(* CODESYS project Motion.library
   Version: 2025.10.15.1
   Title: Motion
   DefaultNamespace: Motion
   Placeholder: Motion
   Company: Photara

Project tree, tasks and I/O mapping:
  libraries: Base, * (Photara); Communication, * (Photara); Tc2_MC2, * (Beckhoff Automation GmbH); Tc2_MC2_Drive, * (Beckhoff Automation GmbH); Tc2_Standard, * (Beckhoff Automation GmbH); Tc2_System, * (Beckhoff Automation GmbH); Tc2_Utilities, * (Beckhoff Automation GmbH); Tc3_Module, * (Beckhoff Automation GmbH); TcUnit, * (www.tcunit.org)
  BeckhoffAxis/
    DUTs/
      data type E_WebDriveState
      data type ST_BeckhoffAxisConfiguration
      data type ST_BeckhoffAxisStatus
    GVLs/
      global variables GC_BeckhoffAxis
      global variables GPL_BeckhoffAxis
    POUs/
      function CalculateVirtualDistance [ST]
      function block FB_BeckhoffAxis [ST]: Halt, MoveRelative, MoveVelocity, PowerOff, PowerOn, ResetAxis, SetBrake, SetTension, Stop, _InitializeReferences, _SetCommandPermIntlkConfiguration, _BeckhoffMotionFBs, _CyclicFlags, _EvaluateCompletionConditions, _UpdateComponentStatus, Busy, P_AxisConfiguration, P_AxisReference, P_InTension, P_Powered, P_RotaryAxisStatus, CyclicLogic
      function block FB_WebDrive [ST]: _CalculateRadius, _InitializeChildrenDependencies, CyclicLogic
    Testing/
  ITFs/
    Motion/
      interface I_CompleteAxis: MoveAbsolute
      interface I_RotaryAxis: P_AxisReference, P_RotaryAxisStatus, Halt, MoveRelative, MoveVelocity, PowerOff, PowerOn, ResetAxis, SetBrake, SetTension, Stop
      interface I_RotaryEncoder: Read
  RotaryEncoder/
    DUTs/
      data type ST_RotaryEncoderConfiguration
      data type ST_RotaryEncoderStatus
    GVLs/
      global variables GC_RotaryEncoder
      global variables GPL_RotaryEncoder
    POUs/
      function block FB_RotaryEncoder [ST]: Read, _InitializeReferences, _SetCommandPermIntlkConfiguration, _EvaluateCompletionConditions, _UpdateComponentStatus, CyclicLogic
  Zaber/
    DUTs/
      data type E_MoveDirection
      data type E_MoveType
      data type ST_ArcParameters
      data type ST_AxisKinematics
      data type ST_SinParameters
      data type ST_WaitingForBits
      data type ST_ZaberCommandConfiguration
      data type ST_ZaberConfiguration
      data type ST_ZaberHMI
      data type ST_ZaberInitTableFW744
      data type ST_ZaberReply
      data type ST_ZaberStatus
    GVLs/
      global variables GC_Zaber
      global variables GPL_Zaber
    POUs/
      Functions/
        function F_ExtractAxisNumber [ST]
        function F_ExtractDataField [ST]
        function F_ExtractDeviceAddress [ST]
        function F_ExtractMessageChecksum [ST]
        function F_ExtractMotionStatus [ST]
        function F_ZaberExtractExecutionResult [ST]
        function F_ZaberExtractWarnFaultFlag [ST]
        function F_ZaberSplitReplyTokensEx [ST]
      function block FB_ZaberAxisCmdConfiguration [ST]: _BuildTables, _Initialize, _InitializeChildrenDependencies, _InitializeReferences, FB_Init, GetIndexByCmdSendString, GetIndexByPOUName, P_CommandConfigurations, P_PermIntlkConfigurations, P_ZaberConfiguration, P_ZaberInitTableFW744
      function block FB_ZaberSerialAxis [ST]: comm_en_ipv4_static, io_cancel_schedule, io_set_ao, io_set_ao_schedule, io_set_do, io_set_do_schedule, lockstep_driver_disable, lockstep_driver_enable, lockstep_move_abs, lockstep_move_rel, lockstep_move_sin_stop, lockstep_move_stored, lockstep_move_vel, lockstep_park, lockstep_print, lockstep_set_tolerance, lockstep_setup_disable, lockstep_setup_enable, lockstep_stop, lockstep_unpark, move_index, move_rel, move_sin_stop, move_stored, pvt_buffer_erase, pvt_buffer_print, pvt_call, pvt_fifo, pvt_info, pvt_io_cancel_schedule, pvt_io_set_ao, pvt_io_set_ao_schedule, pvt_io_set_do, pvt_io_set_do_schedule, pvt_point, pvt_setup_disable, pvt_setup_live, pvt_setup_store, scope_add, scope_add_io_ai, scope_add_io_ao, scope_add_io_di, scope_add_io_do, scope_start, set_accel, set_autodetect_coil_mode, set_calibration_type, set_comm_address, set_comm_alert, set_comm_command_packets_max, set_comm_en_ipv4_address, set_comm_en_ipv4_dhcp_enabled, set_comm_en_ipv4_gateway, set_comm_en_ipv4_netmask, set_comm_en_mac, set_comm_en_mdns_enable, set_comm_next_owner, set_comm_packet_size_max, set_comm_protocol, set_comm_rs232_baud, set_comm_word_size_max, set_driver_current_approach, set_driver_current_hold, set_driver_current_max, set_driver_current_run, set_driver_enable_mode, set_driver_enabled, set_driver_temperature, set_get_settings_max, set_ictrl_advance_a, set_ictrl_advance_offset, set_ictrl_afcff_inductance, set_ictrl_afcff_ke, set_ictrl_afcff_ki, set_ictrl_afcff_max, set_ictrl_afcff_ss, set_ictrl_afcff_ss_max, set_ictrl_delay, set_ictrl_ff_kd, set_ictrl_ff_kp, set_ictrl_gain_coldmult, set_ictrl_period, set_ictrl_pi_ki, set_ictrl_pi_kp, set_ictrl_type, set_io_ai_1_fc, set_io_ai_2_fc, set_io_ai_3_fc, set_io_ai_4_fc, set_io_di_port, set_io_do_port, set_knob_dir, set_knob_distance, set_knob_enable, set_knob_maxspeed, set_knob_mode, set_knob_speedprofile, set_limit_approach_maxspeed, set_limit_detect_decelonly, set_limit_detect_maxspeed, set_limit_home_action, set_limit_home_bidirectional, set_limit_home_edge, set_limit_home_offset, set_limit_home_posupdate, set_limit_home_preset, set_limit_home_source, set_limit_home_state, set_limit_home_triggered, set_limit_home_tune, set_limit_home_type, set_limit_home_width, set_limit_max, set_limit_min, set_limit_range_mode, set_lockstep_numgroups, set_maxspeed, set_motion_accel_ramptime, set_motion_accelonly, set_motion_busy, set_motion_decelonly, set_motion_index_dist, set_motion_index_num, set_motion_tracking_ai, set_motion_tracking_dir, set_motion_tracking_ki, set_motion_tracking_kp, set_motion_tracking_limit_max, set_motion_tracking_limit_min, set_motion_tracking_scan_dir, set_motion_tracking_scan_maxspeed, set_motion_tracking_scan_offset, set_motion_tracking_scan_period, set_motion_tracking_scan_signal_valid_delay, set_motion_tracking_scan_tolerance, set_motion_tracking_setpoint, set_motion_tracking_settle_period, set_motion_tracking_settle_tolerance, set_motion_tracking_settle_tolerance_met, set_motion_tracking_settled, set_motion_tracking_signal_valid_di, set_motor_current_max, set_motor_inductance, set_motor_ke, set_motor_phase, set_motor_phase_ratio_div1, set_motor_phase_ratio_div2, set_motor_phase_ratio_mult, set_motor_resistance, set_parking_state, set_peripheral_hw_modified, set_peripheral_id, set_peripheral_id_pending, set_peripheral_serial, set_peripheral_serial_pending, set_pos, set_pvt_numseqs, set_resolution, set_scope_channel_size, set_scope_channel_size_max, set_scope_delay, set_scope_numchannels, set_scope_timebase, set_stream_numbufs, set_stream_numstreams, set_system_access, set_system_axiscount, set_system_led_enable, set_system_serial, set_system_temperature, set_system_uptime, set_system_voltage, set_trigger_numactions, set_trigger_numtriggers, set_user_data_0, set_user_data_1, set_user_data_10, set_user_data_11, set_user_data_12, set_user_data_13, set_user_data_14, set_user_data_15, set_user_data_2, set_user_data_3, set_user_data_4, set_user_data_5, set_user_data_6, set_user_data_7, set_user_data_8, set_user_data_9, set_user_vdata_0, set_user_vdata_1, set_user_vdata_2, set_user_vdata_3, set_vel, set_version, set_version_build, storage_append, storage_exists, storage_get, storage_set, stream_arc, stream_buffer_erase, stream_buffer_print, stream_call, stream_circle, stream_fifo, stream_helix, stream_hold_onloff, stream_info, stream_io_cancel_schedule, stream_io_set_ao, stream_io_set_ao_schedule, stream_io_set_do, stream_io_set_do_schedule, stream_line, stream_set, stream_setup_disable, stream_setup_live, stream_setup_store, stream_wait, stream_wait_io, tools_storepos, trigger_action_command, trigger_action_none, trigger_action_setting, trigger_disable, trigger_enable, trigger_when_io, trigger_when_setting, trigger_when_time, activate, axis_restore, comm_en_ipv4_dhcp, driver_disable, driver_enable, get_accel, get_autodetect_coil_mode, get_calibration_type, get_comm_address, get_comm_alert, get_comm_checksum, get_comm_command_packets_max, get_comm_en_ipv4_address, get_comm_en_ipv4_dhcp_enabled, get_comm_en_ipv4_gateway, get_comm_en_ipv4_netmask, get_comm_en_mac, get_comm_en_mdns_enable, get_comm_next_owner, get_comm_packet_size_max, get_comm_protocol, get_comm_rs232_baud, get_comm_word_size_max, get_device_hw_modified, get_device_id, get_driver_current_approach, get_driver_current_hold, get_driver_current_max, get_driver_current_run, get_driver_enable_mode, get_driver_enabled, get_driver_temperature, get_get_settings_max, get_ictrl_advance_a, get_ictrl_advance_offset, get_ictrl_afcff_inductance, get_ictrl_afcff_ke, get_ictrl_afcff_ki, get_ictrl_afcff_max, get_ictrl_afcff_ss, get_ictrl_afcff_ss_max, get_ictrl_delay, get_ictrl_ff_kd, get_ictrl_ff_kp, get_ictrl_gain_coldmult, get_ictrl_period, get_ictrl_pi_ki, get_ictrl_pi_kp, get_ictrl_type, get_io_ai_1_fc, get_io_ai_2_fc, get_io_ai_3_fc, get_io_ai_4_fc, get_io_di_port, get_io_do_port, get_knob_dir, get_knob_distance, get_knob_enable, get_knob_maxspeed, get_knob_mode, get_knob_speedprofile, get_limit_approach_maxspeed, get_limit_detect_decelonly, get_limit_detect_maxspeed, get_limit_home_action, get_limit_home_bidirectional, get_limit_home_edge, get_limit_home_offset, get_limit_home_posupdate, get_limit_home_preset, get_limit_home_source, get_limit_home_state, get_limit_home_triggered, get_limit_home_tune, get_limit_home_type, get_limit_home_width, get_limit_max, get_limit_min, get_limit_range_mode, get_lockstep_numgroups, get_maxspeed, get_motion_accel_ramptime, get_motion_accelonly, get_motion_busy, get_motion_decelonly, get_motion_index_dist, get_motion_index_num, get_motion_tracking_ai, get_motion_tracking_dir, get_motion_tracking_ki, get_motion_tracking_kp, get_motion_tracking_limit_max, get_motion_tracking_limit_min, get_motion_tracking_scan_dir, get_motion_tracking_scan_maxspeed, get_motion_tracking_scan_offset, get_motion_tracking_scan_period, get_motion_tracking_scan_signal_valid_delay, get_motion_tracking_scan_tolerance, get_motion_tracking_setpoint, get_motion_tracking_settle_period, get_motion_tracking_settle_tolerance, get_motion_tracking_settle_tolerance_met, get_motion_tracking_settled, get_motion_tracking_signal_valid_di, get_motor_current_max, get_motor_inductance, get_motor_ke, get_motor_phase, get_motor_phase_ratio_div1, get_motor_phase_ratio_div2, get_motor_phase_ratio_mult, get_motor_resistance, get_parking_state, get_peripheral_hw_modified, get_peripheral_id, get_peripheral_id_pending, get_peripheral_serial, get_peripheral_serial_pending, get_pos, get_pvt_numseqs, get_resolution, get_scope_channel_size, get_scope_channel_size_max, get_scope_delay, get_scope_numchannels, get_scope_timebase, get_stream_numbufs, get_stream_numstreams, get_system_access, get_system_axiscount, get_system_current_max, get_system_led_enable, get_system_serial, get_system_temperature, get_system_uptime, get_system_voltage, get_trigger_numactions, get_trigger_numtriggers, get_user_data_0, get_user_data_1, get_user_data_10, get_user_data_11, get_user_data_12, get_user_data_13, get_user_data_14, get_user_data_15, get_user_data_2, get_user_data_3, get_user_data_4, get_user_data_5, get_user_data_6, get_user_data_7, get_user_data_8, get_user_data_9, get_user_vdata_0, get_user_vdata_1, get_user_vdata_2, get_user_vdata_3, get_vel, get_version, get_version_build, home, io_get_ai, io_get_ao, io_get_di, io_get_do, io_info, lockstep_get, lockstep_home, lockstep_move_max, lockstep_move_min, lockstep_move_sin, move_abs, move_index_next, move_index_prev, move_max, move_min, move_scan_track_once, move_sin, move_track, move_vel, pvt_buffer_list, renumber, scope_clear, scope_print, scope_stop, set_comm_checksum, stop, storage_erase, storage_print, stream_buffer_list, system_errors, system_factoryreset, system_reset, system_restore, tools_echo, tools_findrange, tools_gotolimit, tools_parking, tools_setcomm, tools_storepos_current, tools_storepos_position, trigger_print, trigger_show, trigger_when_dist, trigger_when_encoder_dist, warnings, warnings_clear, CyclicLogic, P_ZaberConfiguration, _Initialize, _InitializeChildrenDependencies, _InitializeReferences, FB_Init, InjectDependencies, _BuildCommandStringNoArgs, _ClearTempString, _ConfigurationCyclic, _DebugTesting, _DispatchValid, _GetConfigParametersOnInit, _MapIndicesToCommands, _MonitorAsynchronousRequests, _PollBusy, _PopulateStatusStructureWithResponseData, _ReceiveCyclic, _ResolveZaberConfiguration, _ResolveZaberDispatchIndex, _SendCyclic, _TryRehashDispatchIndex, _ExecuteCommandByIndexCyclic, ExecuteCommand, InjectConfigurations, P_I_RingBufferKeyString
      function block FB_ZaberSerialGroup [ST]: _ControllerAxisConfiguration, _Initialize, _InitializeChildrenDependencies, CyclicLogic, FB_Init
    Testing/
      function block FB_ValidateStringHandlingTests [ST]: GivenBusyReplyExpectCorrectFieldExtractionChecksum, GivenBusyReplyExpectCorrectFieldExtractionNoChecksum, GivenIdleReplyExpectCorrectFieldExtractionChecksum, GivenIdleReplyExpectCorrectFieldExtractionChecksum_1, GivenIdleReplyExpectCorrectFieldExtractionNoChecksum, GivenNIReplyExpectCorrectFieldExtractionChecksum, GivenNIReplyExpectCorrectFieldExtractionNoChecksum, GivenReply_ExpectCorrectTokenization
      function block FB_ZaberAxisTests [ST]
      program PRG_TEST [ST]
  program MAIN [ST]
*)

// BeckhoffAxis/DUTs/E_WebDriveState
{attribute 'qualified_only'}
{attribute 'strict'}
{attribute 'to_string'}
TYPE E_WebDriveState :
(
	INIT := 0,
	STOP,
	RESET,
	ERROR,
	IDLE,
	BUSY_TENSION,
	BUSY_SCROLL,
	CALIBRATION
);
END_TYPE

// BeckhoffAxis/DUTs/ST_BeckhoffAxisConfiguration
TYPE ST_BeckhoffAxisConfiguration :
STRUCT
	ComponentConfiguration : REFERENCE TO Base.ST_ComponentConfiguration;
	
	lrTorqueRamp : LREAL := 3; // Tensies per second
	lrMaxSpeed	 : LREAL := 2_000.0; // mm/s
	
	lrScrollVelocity : LREAL := 400.0; // mm/s
END_STRUCT
END_TYPE

// BeckhoffAxis/DUTs/ST_BeckhoffAxisStatus
TYPE ST_BeckhoffAxisStatus :
STRUCT
	BaseComponentStatus : REFERENCE TO Base.ST_ComponentStatus;
	
END_STRUCT
END_TYPE

// RotaryEncoder/DUTs/ST_RotaryEncoderConfiguration
TYPE ST_RotaryEncoderConfiguration :
STRUCT
	ComponentConfiguration : REFERENCE TO Base.ST_ComponentConfiguration;
	CPmm : REAL := 13.123; // clicks on encoder per mm travelled
END_STRUCT
END_TYPE

// RotaryEncoder/DUTs/ST_RotaryEncoderStatus
TYPE ST_RotaryEncoderStatus :
STRUCT
	BaseComponentStatus : REFERENCE TO Base.ST_ComponentStatus;
END_STRUCT
END_TYPE

// Zaber/DUTs/E_MoveDirection
{attribute 'qualified_only'}
{attribute 'strict'}
{attribute 'to_string'}
TYPE E_MoveDirection :
(
	cw := 0, //clockwise
	ccw := 1 //counter-clockwise
);
END_TYPE

// Zaber/DUTs/E_MoveType
{attribute 'qualified_only'}
{attribute 'strict'}
{attribute 'to_string'}
TYPE E_MoveType :
(
	move_abs := 0,
	move_rel := 1
);
END_TYPE

// Zaber/DUTs/ST_ArcParameters
TYPE ST_ArcParameters :
STRUCT
	Axis1 : UINT; //<axis1> The first stream axis on which TO execute the arc segment (optional).  The first stream axis is labelled "a", the second "b", AND so on
	Axis2 : UINT; //<axis2> The second stream axis on which to execute the arc segment (optional). The first stream axis is labelled "a", the second "b", and so on
	MoveType : E_MoveType; //abs Indicates that position parameters are absolute positions; rel Indicates that position parameters are relative to the end point of the previous path segment
	Direction : E_MoveDirection; //cw Indicates that the arc should be in the clockwise direction; //ccw Indicates that the arc should be in the counter-clockwise direction
	CenterX : DINT; //<centrex> The x-axis position of the arc’s centre; Must be the range -2,147,483,648 to 2,147,483,647
	CenterY : DINT; //<centrey> The y-axis position of the arc’s centre; Must be the range -2,147,483,648 to 2,147,483,647
	EndX : DINT; //<endx> The x-axis position of the end of the arc; Must be in the range limit.min to limit.max for that axis
	EndY : DINT; //<endy> The y-axis position of the end of the arc; Must be in the range limit.min to limit.max for that axis
END_STRUCT
END_TYPE

// Zaber/DUTs/ST_AxisKinematics
TYPE ST_AxisKinematics :
STRUCT
	Position	: UDINT;
	Velocity	: DINT;
	Accel		: UDINT;
END_STRUCT
END_TYPE

// Zaber/DUTs/ST_SinParameters
TYPE ST_SinParameters :
STRUCT
	Amplitude					: LREAL := 50000;
	Period						: LREAL := 2000; // ms
	Count						: LREAL := 30;
END_STRUCT
END_TYPE

// Zaber/DUTs/ST_WaitingForBits
TYPE ST_WaitingForBits :
STRUCT
	WaitingForResolution	: BOOL;
	WaitingForMaxSpeed		: BOOL;
END_STRUCT
END_TYPE

// Zaber/DUTs/ST_ZaberCommandConfiguration
TYPE ST_ZaberCommandConfiguration :
STRUCT
 //   CmdIndex			: DINT; 
    PouName 			: STRING;
    CmdDesc				: STRING;
	CmdExecutionType	: Base.E_CommandExecutionType;
END_STRUCT
END_TYPE

// Zaber/DUTs/ST_ZaberConfiguration
TYPE ST_ZaberConfiguration :
STRUCT
	ComponentConfiguration 			: REFERENCE TO ST_ComponentConfiguration;
	ConfiguredComPort				: UDINT := 3;
	ConfiguredTerminationTx			: STRING(5) := '$N';
	ConfiguredTerminationRx			: STRING(5) := '$R$N';
	sControllerRef					: STRING(5) := '/0';
	AxisRef							: UINT := 0;
	MinDynamics						: ST_AxisKinematics;
	MaxDynamics						: ST_AxisKinematics := (Position := 227000, Velocity := 100000, Accel := 15000);
	SetDynamics						: ST_AxisKinematics := (Position := 113000, Velocity := MaxDynamics.Velocity, Accel := MaxDynamics.Accel);
	MaxPollingTime					: TIME := T#50MS;
	MinPollingTime					: TIME := T#5MS;
	EnableSerialInterface			: BOOL := TRUE;
	PollingIntervalTime				: TIME := T#20MS;
	EnablePollingOnMotion			: BOOL := TRUE;
	Resolution						: REAL; // microstep div
	Resolution_um					: REAL := 1.984375; // µm; given by manual
	StreamNumber					: ARRAY[GPL_Zaber.INDEX_STREAM_MIN..GPL_Zaber.INDEX_STREAM_MAX] OF UDINT; 
	BufferNumber					: UDINT;
	LockstepGroup					: USINT := 1;
	TimeConversionFactor			: REAL := 16.384; //s; given by manual
	EnableDynamicPollingInterval	: BOOL := TRUE;
	DefaultPollingTime				: TIME := T#10MS;
	EnableGetParametersOnInit		: BOOL;
	RelativeDistanceMove			: UDINT := 1000; // µm; 
	SinParameters					: ST_SinParameters;
	ArcParameters					: ST_ArcParameters;
	Direction						: BOOL := TRUE; //Right/CW = TRUE
	GetSetting						: STRING(15) := 'twist';
	OptionalValue					: STRING(GPL_Zaber.STRING_LENGTH);
END_STRUCT
END_TYPE

// Zaber/DUTs/ST_ZaberHMI
TYPE ST_ZaberHMI :
STRUCT
    ReplyFlag		: STRING(GPL_Zaber.STRING_LENGTH);  // 'OK' / 'RJ'
    MotionStatus	: BOOL;  // BUSY / IDLE
    WarnFlag    	: STRING(GPL_Zaber.STRING_LENGTH);  // '--' or 'FV'… or 'NI'
    DataField   	: STRING(GPL_Zaber.STRING_LENGTH);  // '0', '12345', etc.
    Checksum    	: STRING(GPL_Zaber.STRING_LENGTH);  // ':CC' or ''
	Footer			: STRING(GPL_Zaber.STRING_LENGTH);
	Position		: DINT;
	Velocity		: DINT; // parsed from Data Field
END_STRUCT
END_TYPE

// Zaber/DUTs/ST_ZaberInitTableFW744
TYPE ST_ZaberInitTableFW744 :
STRUCT
    CmdIndex        : ARRAY[GC_Zaber.INDEX_COMMAND_MIN..GC_Zaber.INDEX_COMMAND_MAX] OF DINT; 
    PouName : ARRAY[GC_Zaber.INDEX_COMMAND_MIN..GC_Zaber.INDEX_COMMAND_MAX] OF STRING := [
        'activate',
        'axis_restore',
        'driver_disable',
        'driver_enable',
        'home',
        'renumber',
        'stop',
        'warnings',
        'comm_en_ipv4_dhcp',
        'comm_en_ipv4_static',
        'io_cancel_schedule',
        'io_get_ai',
        'io_get_ao',
        'io_get_di',
        'io_get_do',
        'io_info',
        'io_set_ao',
        'io_set_ao_schedule',
        'io_set_do',
        'io_set_do_schedule',
        'move_abs',
        'move_index',
        'move_index_next',
        'move_index_prev',
        'move_min',
        'move_max',
        'move_rel',
        'move_scan_track_once',
        'move_sin',
        'move_sin_stop',
        'move_stored',
        'move_track',
        'move_vel',
        'lockstep_driver_disable',
        'lockstep_driver_enable',
        'lockstep_get',
        'lockstep_home',
        'lockstep_move_abs',
        'lockstep_move_min',
        'lockstep_move_max',
        'lockstep_move_rel',
        'lockstep_move_sin',
        'lockstep_move_sin_stop',
        'lockstep_move_stored',
        'lockstep_move_vel',
        'lockstep_park',
        'lockstep_unpark',
        'lockstep_print',
        'lockstep_set_tolerance',
        'lockstep_setup_disable',
        'lockstep_setup_enable',
        'lockstep_stop',
        'pvt_buffer_erase',
        'pvt_buffer_list',
        'pvt_buffer_print',
        'pvt_call',
        'pvt_fifo',
        'pvt_info',
        'pvt_io_cancel_schedule',
        'pvt_io_set_ao',
        'pvt_io_set_ao_schedule',
        'pvt_io_set_do',
        'pvt_io_set_do_schedule',
        'pvt_point',
        'pvt_setup_disable',
        'pvt_setup_live',
        'pvt_setup_store',
        'scope_add',
        'scope_add_io_ai',
        'scope_add_io_ao',
        'scope_add_io_di',
        'scope_add_io_do',
        'scope_clear',
        'scope_print',
        'scope_start',
        'scope_stop',
        'storage_append',
        'storage_erase',
        'storage_exists',
        'storage_get',
        'storage_print',
        'storage_set',
        'stream_arc',
        'stream_buffer_erase',
        'stream_buffer_list',
        'stream_buffer_print',
        'stream_call',
        'stream_circle',
        'stream_fifo',
        'stream_helix',
        'stream_hold_onloff',
        'stream_info',
        'stream_io_cancel_schedule',
        'stream_io_set_ao',
        'stream_io_set_ao_schedule',
        'stream_io_set_do',
        'stream_io_set_do_schedule',
        'stream_line',
        'stream_set',
        'stream_setup_disable',
        'stream_setup_live',
        'stream_setup_store',
        'stream_wait',
        'stream_wait_io',
        'system_errors',
        'system_factoryreset',
        'system_reset',
        'system_restore',
        'tools_echo',
        'tools_findrange',
        'tools_gotolimit',
        'tools_parking',
        'tools_setcomm',
        'tools_storepos',
        'tools_storepos_current',
        'tools_storepos_position',
        'trigger_action_command',
        'trigger_action_none',
        'trigger_action_setting',
        'trigger_disable',
        'trigger_enable',
        'trigger_print',
        'trigger_show',
        'trigger_when_encoder_dist',
        'trigger_when_dist',
        'trigger_when_io',
        'trigger_when_setting',
        'trigger_when_time',
        'get_accel',
        'get_autodetect_coil_mode',
        'get_calibration_type',
        'get_comm_address',
        'get_comm_alert',
        'get_comm_checksum',
        'get_comm_command_packets_max',
        'get_comm_en_ipv4_address',
        'get_comm_en_ipv4_dhcp_enabled',
        'get_comm_en_ipv4_gateway',
        'get_comm_en_ipv4_netmask',
        'get_comm_en_mac',
        'get_comm_en_mdns_enable',
        'get_comm_next_owner',
        'get_comm_packet_size_max',
        'get_comm_protocol',
        'get_comm_rs232_baud',
        'get_comm_word_size_max',
        'get_device_hw_modified',
        'get_device_id',
        'get_driver_current_approach',
        'get_driver_current_hold',
        'get_driver_current_max',
        'get_driver_current_run',
        'get_driver_enable_mode',
        'get_driver_enabled',
        'get_driver_temperature',
        'get_get_settings_max',
        'get_ictrl_advance_a',
        'get_ictrl_advance_offset',
        'get_ictrl_afcff_inductance',
        'get_ictrl_afcff_ke',
        'get_ictrl_afcff_ki',
        'get_ictrl_afcff_max',
        'get_ictrl_afcff_ss',
        'get_ictrl_afcff_ss_max',
        'get_ictrl_delay',
        'get_ictrl_ff_kd',
        'get_ictrl_ff_kp',
        'get_ictrl_gain_coldmult',
        'get_ictrl_period',
        'get_ictrl_pi_ki',
        'get_ictrl_pi_kp',
        'get_ictrl_type',
        'get_io_ai_1_fc',
        'get_io_ai_2_fc',
        'get_io_ai_3_fc',
        'get_io_ai_4_fc',
        'get_io_di_port',
        'get_io_do_port',
        'get_knob_dir',
        'get_knob_distance',
        'get_knob_enable',
        'get_knob_maxspeed',
        'get_knob_mode',
        'get_knob_speedprofile',
        'get_limit_approach_maxspeed',
        'get_limit_detect_decelonly',
        'get_limit_detect_maxspeed',
        'get_limit_home_action',
        'get_limit_home_bidirectional',
        'get_limit_home_edge',
        'get_limit_home_offset',
        'get_limit_home_posupdate',
        'get_limit_home_preset',
        'get_limit_home_source',
        'get_limit_home_state',
        'get_limit_home_triggered',
        'get_limit_home_tune',
        'get_limit_home_type',
        'get_limit_home_width',
        'get_limit_max',
        'get_limit_min',
        'get_limit_range_mode',
        'get_lockstep_numgroups',
        'get_maxspeed',
        'get_motion_accel_ramptime',
        'get_motion_accelonly',
        'get_motion_busy',
        'get_motion_decelonly',
        'get_motion_index_dist',
        'get_motion_index_num',
        'get_motion_tracking_ai',
        'get_motion_tracking_dir',
        'get_motion_tracking_ki',
        'get_motion_tracking_kp',
        'get_motion_tracking_limit_max',
        'get_motion_tracking_limit_min',
        'get_motion_tracking_scan_dir',
        'get_motion_tracking_scan_maxspeed',
        'get_motion_tracking_scan_offset',
        'get_motion_tracking_scan_period',
        'get_motion_tracking_scan_signal_valid_delay',
        'get_motion_tracking_scan_tolerance',
        'get_motion_tracking_setpoint',
        'get_motion_tracking_settle_period',
        'get_motion_tracking_settle_tolerance',
        'get_motion_tracking_settle_tolerance_met',
        'get_motion_tracking_settled',
        'get_motion_tracking_signal_valid_di',
        'get_motor_current_max',
        'get_motor_inductance',
        'get_motor_ke',
        'get_motor_phase',
        'get_motor_phase_ratio_div1',
        'get_motor_phase_ratio_div2',
        'get_motor_phase_ratio_mult',
        'get_motor_resistance',
        'get_parking_state',
        'get_peripheral_hw_modified',
        'get_peripheral_id',
        'get_peripheral_id_pending',
        'get_peripheral_serial',
        'get_peripheral_serial_pending',
        'get_pos',
        'get_pvt_numseqs',
        'get_resolution',
        'get_scope_channel_size',
        'get_scope_channel_size_max',
        'get_scope_delay',
        'get_scope_numchannels',
        'get_scope_timebase',
        'get_stream_numbufs',
        'get_stream_numstreams',
        'get_system_access',
        'get_system_axiscount',
        'get_system_current_max',
        'get_system_led_enable',
        'get_system_serial',
        'get_system_temperature',
        'get_system_uptime',
        'get_system_voltage',
        'get_trigger_numactions',
        'get_trigger_numtriggers',
        'get_user_data_0',
        'get_user_data_1',
        'get_user_data_10',
        'get_user_data_11',
        'get_user_data_12',
        'get_user_data_13',
        'get_user_data_14',
        'get_user_data_15',
        'get_user_data_2',
        'get_user_data_3',
        'get_user_data_4',
        'get_user_data_5',
        'get_user_data_6',
        'get_user_data_7',
        'get_user_data_8',
        'get_user_data_9',
        'get_user_vdata_0',
        'get_user_vdata_1',
        'get_user_vdata_2',
        'get_user_vdata_3',
        'get_vel',
        'get_version',
        'get_version_build',
        'set_accel',
        'set_autodetect_coil_mode',
        'set_calibration_type',
        'set_comm_address',
        'set_comm_alert',
        'set_comm_checksum',
        'set_comm_command_packets_max',
        'set_comm_en_ipv4_address',
        'set_comm_en_ipv4_dhcp_enabled',
        'set_comm_en_ipv4_gateway',
        'set_comm_en_ipv4_netmask',
        'set_comm_en_mdns_enable',
        'set_comm_en_mac',
        'set_comm_next_owner',
        'set_comm_packet_size_max',
        'set_comm_protocol',
        'set_comm_rs232_baud',
        'set_comm_word_size_max',
        'set_driver_current_approach',
        'set_driver_current_hold',
        'set_driver_current_max',
        'set_driver_current_run',
        'set_driver_enable_mode',
        'set_driver_enabled',
        'set_driver_temperature',
        'set_get_settings_max',
        'set_ictrl_advance_a',
        'set_ictrl_advance_offset',
        'set_ictrl_afcff_inductance',
        'set_ictrl_afcff_ke',
        'set_ictrl_afcff_ki',
        'set_ictrl_afcff_max',
        'set_ictrl_afcff_ss',
        'set_ictrl_afcff_ss_max',
        'set_ictrl_delay',
        'set_ictrl_ff_kd',
        'set_ictrl_ff_kp',
        'set_ictrl_gain_coldmult',
        'set_ictrl_period',
        'set_ictrl_pi_ki',
        'set_ictrl_pi_kp',
        'set_ictrl_type',
        'set_io_ai_1_fc',
        'set_io_ai_2_fc',
        'set_io_ai_3_fc',
        'set_io_ai_4_fc',
        'set_io_di_port',
        'set_io_do_port',
        'set_knob_dir',
        'set_knob_distance',
        'set_knob_enable',
        'set_knob_maxspeed',
        'set_knob_mode',
        'set_knob_speedprofile',
        'set_limit_approach_maxspeed',
        'set_limit_detect_decelonly',
        'set_limit_detect_maxspeed',
        'set_limit_home_action',
        'set_limit_home_bidirectional',
        'set_limit_home_edge',
        'set_limit_home_offset',
        'set_limit_home_posupdate',
        'set_limit_home_preset',
        'set_limit_home_source',
        'set_limit_home_state',
        'set_limit_home_triggered',
        'set_limit_home_tune',
        'set_limit_home_type',
        'set_limit_home_width',
        'set_limit_max',
        'set_limit_min',
        'set_limit_range_mode',
        'set_lockstep_numgroups',
        'set_maxspeed',
        'set_motion_accel_ramptime',
        'set_motion_accelonly',
        'set_motion_busy',
        'set_motion_decelonly',
        'set_motion_index_dist',
        'set_motion_index_num',
        'set_motion_tracking_ai',
        'set_motion_tracking_dir',
        'set_motion_tracking_ki',
        'set_motion_tracking_kp',
        'set_motion_tracking_limit_max',
        'set_motion_tracking_limit_min',
        'set_motion_tracking_scan_dir',
        'set_motion_tracking_scan_maxspeed',
        'set_motion_tracking_scan_offset',
        'set_motion_tracking_scan_period',
        'set_motion_tracking_scan_signal_valid_delay',
        'set_motion_tracking_scan_tolerance',
        'set_motion_tracking_setpoint',
        'set_motion_tracking_settle_period',
        'set_motion_tracking_settle_tolerance',
        'set_motion_tracking_settle_tolerance_met',
        'set_motion_tracking_settled',
        'set_motion_tracking_signal_valid_di',
        'set_motor_current_max',
        'set_motor_inductance',
        'set_motor_ke',
        'set_motor_phase',
        'set_motor_phase_ratio_div1',
        'set_motor_phase_ratio_div2',
        'set_motor_phase_ratio_mult',
        'set_motor_resistance',
        'set_parking_state',
        'set_peripheral_hw_modified',
        'set_peripheral_id',
        'set_peripheral_id_pending',
        'set_peripheral_serial',
        'set_peripheral_serial_pending',
        'set_pos',
        'set_pvt_numseqs',
        'set_resolution',
        'set_scope_channel_size',
        'set_scope_channel_size_max',
        'set_scope_delay',
        'set_scope_numchannels',
        'set_scope_timebase',
        'set_stream_numbufs',
        'set_stream_numstreams',
        'set_system_access',
        'set_system_axiscount',
        'set_system_led_enable',
        'set_system_serial',
        'set_system_temperature',
        'set_system_uptime',
        'set_system_voltage',
        'set_trigger_numactions',
        'set_trigger_numtriggers',
        'set_user_data_0',
        'set_user_data_1',
        'set_user_data_2',
        'set_user_data_3',
        'set_user_data_4',
        'set_user_data_5',
        'set_user_data_6',
        'set_user_data_7',
        'set_user_data_8',
        'set_user_data_9',
        'set_user_data_10',
        'set_user_data_11',
        'set_user_data_12',
        'set_user_data_13',
        'set_user_data_14',
        'set_user_data_15',
        'set_user_vdata_0',
        'set_user_vdata_1',
        'set_user_vdata_2',
        'set_user_vdata_3',
        'set_vel',
        'set_version',
        'set_version_build',
		'warnings_clear'
    ];
    
    CmdDesc : ARRAY[GC_Zaber.INDEX_COMMAND_MIN..GC_Zaber.INDEX_COMMAND_MAX] OF STRING := [
        'activate',
        'axis restore',
        'driver disable',
        'driver enable',
        'home',
        'renumber',
        'stop',
        'warnings',
        'comm en ipv4 dhcp',
        'comm en ipv4 static',
        'io cancel schedule',
        'io get ai',
        'io get ao',
        'io get di',
        'io get do',
        'io info',
        'io set ao',
        'io set ao schedule',
        'io set do',
        'io set do schedule',
        'move abs',
        'move index',
        'move index next',
        'move index prev',
        'move min',
        'move max',
        'move rel',
        'move scan track once',
        'move sin',
        'move sin stop',
        'move stored',
        'move track',
        'move vel',
        'lockstep driver disable', // note - string parsed in method
        'lockstep driver enable',
        'lockstep get',
        'lockstep home',
        'lockstep move abs',
        'lockstep move min',
        'lockstep move max',
        'lockstep move rel',
        'lockstep move sin',
        'lockstep move sin stop',
        'lockstep move stored',
        'lockstep move vel',
        'lockstep park',
        'lockstep unpark',
        'lockstep print',
        'lockstep set tolerance',
        'lockstep setup disable',
        'lockstep setup enable',
        'lockstep stop',
        'pvt buffer erase',
        'pvt buffer list',
        'pvt buffer print',
        'pvt call',
        'pvt fifo',
        'pvt info',
        'pvt io cancel schedule',
        'pvt io set ao',
        'pvt io set ao schedule',
        'pvt io set do',
        'pvt io set do schedule',
        'pvt point',
        'pvt setup disable',
        'pvt setup live',
        'pvt setup store',
        'scope add',
        'scope add io ai',
        'scope add io ao',
        'scope add io di',
        'scope add io do',
        'scope clear',
        'scope print',
        'scope start',
        'scope stop',
        'storage append',
        'storage erase',
        'storage exists',
        'storage get',
        'storage print',
        'storage set',
        'stream arc',
        'stream buffer erase',
        'stream buffer list',
        'stream buffer print',
        'stream call',
        'stream circle',
        'stream fifo',
        'stream helix',
        'stream hold onloff',
        'stream info',
        'stream io cancel schedule',
        'stream io set ao',
        'stream io set ao schedule',
        'stream io set do',
        'stream io set do schedule',
        'stream line',
        'stream set',
        'stream setup disable',
        'stream setup live',
        'stream setup store',
        'stream wait',
        'stream wait io',
        'system errors',
        'system factoryreset',
        'system reset',
        'system restore',
        'tools echo',
        'tools findrange',
        'tools gotolimit',
        'tools parking',
        'tools setcomm',
        'tools storepos',
        'tools storepos current',
        'tools storepos position',
        'trigger action command',
        'trigger action none',
        'trigger action setting',
        'trigger disable',
        'trigger enable',
        'trigger print',
        'trigger show',
        'trigger when encoder dist',
        'trigger when dist',
        'trigger when io',
        'trigger when setting',
        'trigger when time',
        'get accel',
        'get autodetect.coil.mode',
        'get calibration.type',
        'get comm.address',
        'get comm.alert',
        'get comm.checksum',
        'get comm.command.packets.max',
        'get comm.en.ipv4.address',
        'get comm.en.ipv4.dhcp.enabled',
        'get comm.en.ipv4.gateway',
        'get comm.en.ipv4.netmask',
        'get comm.en.mac',
        'get comm.en.mdns.enable',
        'get comm.next.owner',
        'get comm.packet.size.max',
        'get comm.protocol',
        'get comm.rs232.baud',
        'get comm.word.size.max',
        'get device.hw.modified',
        'get device.id',
        'get driver.current.approach',
        'get driver.current.hold',
        'get driver.current.max',
        'get driver.current.run',
        'get driver.enable.mode',
        'get driver.enabled',
        'get driver.temperature',
        'get get.settings.max',
        'get ictrl.advance.a',
        'get ictrl.advance.offset',
        'get ictrl.afcff.inductance',
        'get ictrl.afcff.ke',
        'get ictrl.afcff.ki',
        'get ictrl.afcff.max',
        'get ictrl.afcff.ss',
        'get ictrl.afcff.ss.max',
        'get ictrl.delay',
        'get ictrl.ff.kd',
        'get ictrl.ff.kp',
        'get ictrl.gain.coldmult',
        'get ictrl.period',
        'get ictrl.pi.ki',
        'get ictrl.pi.kp',
        'get ictrl.type',
        'get io.ai.1.fc',
        'get io.ai.2.fc',
        'get io.ai.3.fc',
        'get io.ai.4.fc',
        'get io.di.port',
        'get io.do.port',
        'get knob.dir',
        'get knob.distance',
        'get knob.enable',
        'get knob.maxspeed',
        'get knob.mode',
        'get knob.speedprofile',
        'get limit.approach.maxspeed',
        'get limit.detect.decelonly',
        'get limit.detect.maxspeed',
        'get limit.home.action',
        'get limit.home.bidirectional',
        'get limit.home.edge',
        'get limit.home.offset',
        'get limit.home.posupdate',
        'get limit.home.preset',
        'get limit.home.source',
        'get limit.home.state',
        'get limit.home.triggered',
        'get limit.home.tune',
        'get limit.home.type',
        'get limit.home.width',
        'get limit.max',
        'get limit.min',
        'get limit.range.mode',
        'get lockstep.numgroups',
        'get maxspeed',
        'get motion.accel.ramptime',
        'get motion.accelonly',
        'get motion.busy',
        'get motion.decelonly',
        'get motion.index.dist',
        'get motion.index.num',
        'get motion.tracking.ai',
        'get motion.tracking.dir',
        'get motion.tracking.ki',
        'get motion.tracking.kp',
        'get motion.tracking.limit.max',
        'get motion.tracking.limit.min',
        'get motion.tracking.scan.dir',
        'get motion.tracking.scan.maxspeed',
        'get motion.tracking.scan.offset',
        'get motion.tracking.scan.period',
        'get motion.tracking.scan.signal.valid.delay',
        'get motion.tracking.scan.tolerance',
        'get motion.tracking.setpoint',
        'get motion.tracking.settle.period',
        'get motion.tracking.settle.tolerance',
        'get motion.tracking.settle.tolerance.met',
        'get motion.tracking.settled',
        'get motion.tracking.signal.valid.di',
        'get motor.current.max',
        'get motor.inductance',
        'get motor.ke',
        'get motor.phase',
        'get motor.phase.ratio.div1',
        'get motor.phase.ratio.div2',
        'get motor.phase.ratio.mult',
        'get motor.resistance',
        'get parking.state',
        'get peripheral.hw.modified',
        'get peripheral.id',
        'get peripheral.id.pending',
        'get peripheral.serial',
        'get peripheral.serial.pending',
        'get pos',
        'get pvt.numseqs',
        'get resolution',
        'get scope.channel.size',
        'get scope.channel.size.max',
        'get scope.delay',
        'get scope.numchannels',
        'get scope.timebase',
        'get stream.numbufs',
        'get stream.numstreams',
        'get system.access',
        'get system.axiscount',
        'get system.current.max',
        'get system.led.enable',
        'get system.serial',
        'get system.temperature',
        'get system.uptime',
        'get system.voltage',
        'get trigger.numactions',
        'get trigger.numtriggers',
        'get user.data.0',
        'get user.data.1',
        'get user.data.10',
        'get user.data.11',
        'get user.data.12',
        'get user.data.13',
        'get user.data.14',
        'get user.data.15',
        'get user.data.2',
        'get user.data.3',
        'get user.data.4',
        'get user.data.5',
        'get user.data.6',
        'get user.data.7',
        'get user.data.8',
        'get user.data.9',
        'get user.vdata.0',
        'get user.vdata.1',
        'get user.vdata.2',
        'get user.vdata.3',
        'get vel',
        'get version',
        'get version.build',
        'set accel',
        'set autodetect.coil.mode',
        'set calibration.type',
        'set comm.address',
        'set comm.alert',
        'set comm.checksum',
        'set comm.command.packets.max',
        'set comm.en.ipv4.address',
        'set comm.en.ipv4.dhcp.enabled',
        'set comm.en.ipv4.gateway',
        'set comm.en.ipv4.netmask',
        'set comm.en.mdns.enable',
        'set comm.en.mac',
        'set comm.next.owner',
        'set comm.packet.size.max',
        'set comm.protocol',
        'set comm.rs232.baud',
        'set comm.word.size.max',
        'set driver.current.approach',
        'set driver.current.hold',
        'set driver.current.max',
        'set driver.current.run',
        'set driver.enable.mode',
        'set driver.enabled',
        'set driver.temperature',
        'set get.settings.max',
        'set ictrl.advance.a',
        'set ictrl.advance.offset',
        'set ictrl.afcff.inductance',
        'set ictrl.afcff.ke',
        'set ictrl.afcff.ki',
        'set ictrl.afcff.max',
        'set ictrl.afcff.ss',
        'set ictrl.afcff.ss.max',
        'set ictrl.delay',
        'set ictrl.ff.kd',
        'set ictrl.ff.kp',
        'set ictrl.gain.coldmult',
        'set ictrl.period',
        'set ictrl.pi.ki',
        'set ictrl.pi.kp',
        'set ictrl.type',
        'set io.ai.1.fc',
        'set io.ai.2.fc',
        'set io.ai.3.fc',
        'set io.ai.4.fc',
        'set io.di.port',
        'set io.do.port',
        'set knob.dir',
        'set knob.distance',
        'set knob.enable',
        'set knob.maxspeed',
        'set knob.mode',
        'set knob.speedprofile',
        'set limit.approach.maxspeed',
        'set limit.detect.decelonly',
        'set limit.detect.maxspeed',
        'set limit.home.action',
        'set limit.home.bidirectional',
        'set limit.home.edge',
        'set limit.home.offset',
        'set limit.home.posupdate',
        'set limit.home.preset',
        'set limit.home.source',
        'set limit.home.state',
        'set limit.home.triggered',
        'set limit.home.tune',
        'set limit.home.type',
        'set limit.home.width',
        'set limit.max',
        'set limit.min',
        'set limit.range.mode',
        'set lockstep.numgroups',
        'set maxspeed',
        'set motion.accel.ramptime',
        'set motion.accelonly',
        'set motion.busy',
        'set motion.decelonly',
        'set motion.index.dist',
        'set motion.index.num',
        'set motion.tracking.ai',
        'set motion.tracking.dir',
        'set motion.tracking.ki',
        'set motion.tracking.kp',
        'set motion.tracking.limit.max',
        'set motion.tracking.limit.min',
        'set motion.tracking.scan.dir',
        'set motion.tracking.scan.maxspeed',
        'set motion.tracking.scan.offset',
        'set motion.tracking.scan.period',
        'set motion.tracking.scan.signal.valid.delay',
        'set motion.tracking.scan.tolerance',
        'set motion.tracking.setpoint',
        'set motion.tracking.settle.period',
        'set motion.tracking.settle.tolerance',
        'set motion.tracking.settle.tolerance.met',
        'set motion.tracking.settled',
        'set motion.tracking.signal.valid.di',
        'set motor.current.max',
        'set motor.inductance',
        'set motor.ke',
        'set motor.phase',
        'set motor.phase.ratio.div1',
        'set motor.phase.ratio.div2',
        'set motor.phase.ratio.mult',
        'set motor.resistance',
        'set parking.state',
        'set peripheral.hw.modified',
        'set peripheral.id',
        'set peripheral.id.pending',
        'set peripheral.serial',
        'set peripheral.serial.pending',
        'set pos',
        'set pvt.numseqs',
        'set resolution',
        'set scope.channel.size',
        'set scope.channel.size.max',
        'set scope.delay',
        'set scope.numchannels',
        'set scope.timebase',
        'set stream.numbufs',
        'set stream.numstreams',
        'set system.access',
        'set system.axiscount',
        'set system.led.enable',
        'set system.serial',
        'set system.temperature',
        'set system.uptime',
        'set system.voltage',
        'set trigger.numactions',
        'set trigger.numtriggers',
        'set user.data.0',
        'set user.data.1',
        'set user.data.2',
        'set user.data.3',
        'set user.data.4',
        'set user.data.5',
        'set user.data.6',
        'set user.data.7',
        'set user.data.8',
        'set user.data.9',
        'set user.data.10',
        'set user.data.11',
        'set user.data.12',
        'set user.data.13',
        'set user.data.14',
        'set user.data.15',
        'set user.vdata.0',
        'set user.vdata.1',
        'set user.vdata.2',
        'set user.vdata.3',
        'set vel',
        'set version',
        'set version.build',
		'warnings clear'
    ];
		CmdExecutionType			: ARRAY[GC_Zaber.INDEX_COMMAND_MIN..GC_Zaber.INDEX_COMMAND_MAX] OF Base.E_CommandExecutionType;
END_STRUCT
END_TYPE

// Zaber/DUTs/ST_ZaberReply
TYPE ST_ZaberReply :
STRUCT
    DeviceAddress	: STRING(GPL_Zaber.STRING_LENGTH);  // '01'
    AxisNumber		: STRING(GPL_Zaber.STRING_LENGTH);  // '0'
    ReplyFlag		: STRING(GPL_Zaber.STRING_LENGTH);  // 'OK' / 'RJ'
    SubCode			: STRING(GPL_Zaber.STRING_LENGTH);  // only if RJ
    MotionStatus	: STRING(GPL_Zaber.STRING_LENGTH);  // BUSY / IDLE
    WarnFlag    	: STRING(GPL_Zaber.STRING_LENGTH);  // '--' or 'FV'… or 'NI'
    DataField   	: STRING(GPL_Zaber.STRING_LENGTH);  // '0', '12345', etc.
    Checksum    	: STRING(GPL_Zaber.STRING_LENGTH);  // ':CC' or ''
	Footer			: STRING(GPL_Zaber.STRING_LENGTH);
END_STRUCT
END_TYPE

// Zaber/DUTs/ST_ZaberStatus
TYPE ST_ZaberStatus :
STRUCT
	ComponentStatus 			: REFERENCE TO ST_ComponentStatus;
	ZaberReply					: ST_ZaberReply;
	ZaberMethodDispatch			: DINT;
	NewResponseParsed			: BOOL;
	ConfigurationResolution		: E_ConfigurationResolution;
	HMIStatus					: ST_ZaberHMI;
	Position					: DINT;
	Velocity					: DINT; // parsed from Data Field
END_STRUCT
END_TYPE

// BeckhoffAxis/GVLs/GC_BeckhoffAxis
{attribute 'qualified_only'}
{attribute 'global_init_slot' := '40622'}
VAR_GLOBAL CONSTANT
	INDEX_COMMAND_MIN : DINT := GPL_BeckhoffAxis.INDEX_COMMAND_MIN;
	INDEX_COMMAND_MAX : DINT := GPL_BeckhoffAxis.INDEX_COMMAND_MAX;
END_VAR

// BeckhoffAxis/GVLs/GPL_BeckhoffAxis
{attribute 'qualified_only'}
{attribute 'global_init_slot' := '40522'}
VAR_GLOBAL CONSTANT
	INDEX_COMMAND_MIN : DINT := 0;
	INDEX_COMMAND_MAX : DINT := 8;
END_VAR

// RotaryEncoder/GVLs/GC_RotaryEncoder
{attribute 'qualified_only'}
{attribute 'global_init_slot' := '41600'}
VAR_GLOBAL CONSTANT
	INDEX_COMMAND_MIN : DINT := GPL_RotaryEncoder.INDEX_COMMAND_MIN;
	INDEX_COMMAND_MAX : DINT := GPL_RotaryEncoder.INDEX_COMMAND_MAX;
END_VAR

// RotaryEncoder/GVLs/GPL_RotaryEncoder
{attribute 'qualified_only'}
{attribute 'global_init_slot' := '41500'}
VAR_GLOBAL CONSTANT
	INDEX_COMMAND_MIN : DINT := 0;
	INDEX_COMMAND_MAX : DINT := 2;
END_VAR

// Zaber/GVLs/GC_Zaber
{attribute 'qualified_only'}
{attribute 'global_init_slot' := '40607'}
VAR_GLOBAL CONSTANT
	INDEX_COMMAND_MIN	: DINT := GPL_Zaber.INDEX_COMMAND_MIN;
	INDEX_COMMAND_MAX	: DINT := GPL_Zaber.INDEX_COMMAND_MAX;
END_VAR

// Zaber/GVLs/GPL_Zaber
{attribute 'qualified_only'}
{attribute 'global_init_slot' := '40507'}
VAR_GLOBAL CONSTANT
	INDEX_COMMAND_MIN			: DINT := 0;
	INDEX_COMMAND_MAX			: DINT := 445;
	STRING_LENGTH 				: USINT := 31;
	
	//Streams
	INDEX_STREAM_MIN			: DINT := 0;
	INDEX_STREAM_MAX			: DINT := 9;
	
	INDEX_AXISGRPINST_MIN		: DINT := 1;
	INDEX_AXISGRPINST_MAX		: DINT := 1;
END_VAR

// BeckhoffAxis/POUs/CalculateVirtualDistance
FUNCTION CalculateVirtualDistance : LREAL
VAR_INPUT
	AngleTurned : LREAL;
	RealDistance : LREAL;
END_VAR
VAR
END_VAR

END_FUNCTION

// BeckhoffAxis/POUs/FB_BeckhoffAxis
FUNCTION_BLOCK FB_BeckhoffAxis EXTENDS Base.FB_Component<GC_BeckhoffAxis.INDEX_COMMAND_MIN,GC_BeckhoffAxis.INDEX_COMMAND_MAX> IMPLEMENTS I_RotaryAxis
VAR CONSTANT
	INDEX_COMMAND_HALT				: DINT := 0;
	INDEX_COMMAND_MOVERELATIVE		: DINT := 1;
	INDEX_COMMAND_MOVEVELOCITY		: DINT := 2;
	INDEX_COMMAND_POWEROFF			: DINT := 3;
	INDEX_COMMAND_POWERON			: DINT := 4;
	INDEX_COMMAND_RESETAXIS			: DINT := 5;
	INDEX_COMMAND_SETBRAKE			: DINT := 6;
	INDEX_COMMAND_SETTENSION		: DINT := 7;
	INDEX_COMMAND_STOP				: DINT := 8;
END_VAR
VAR
	AxisConfiguration 	: ST_BeckhoffAxisConfiguration;
	AxisStatus			: ST_BeckhoffAxisStatus;
	
	lrOverridePower 	: LREAL := 100.0;
	bPowered 			: BOOL;
	bAxisBusy 			: BOOL;

	Axis				: Tc2_MC2.AXIS_REF;
	fbPower	   			: Tc2_MC2.MC_Power;
	fbReset	   			: Tc2_MC2.MC_Reset;
	fbStop				: Tc2_MC2.MC_Stop;
	fbTorque			: Tc2_MC2.MC_TorqueControl;
	fbVelocity			: Tc2_MC2.MC_MoveVelocity;
	fbRelative			: Tc2_MC2.MC_MoveRelative;
	fbHalt				: Tc2_MC2.MC_Halt;
	fbBrakeControl		: Tc2_MC2_Drive.FB_BrakeControl;
	
	bPowerOn 			: BOOL;
	bTorqueFlag			: BOOL;
	bResetFlag			: BOOL;
	bStopFlag			: BOOL;
	bVelocityFlag		: BOOL;
	bRelativeFlag		: BOOL;
	bHaltFlag			: BOOL;
	bBrakeControlFlag	: BOOL;
	
	lrRelDistance		: LREAL;
	lrRelVelocity		: LREAL;
	
	eVelDirection		: MC_Direction := MC_Positive_Direction;
	lrVelVelocity		: LREAL;
	
	eAxisBrakeMode		:  Tc2_MC2_Drive.E_BrakeMode := .E_BrakeMode.eBrakeMode_Automatic;
	
	lrTorqueTensies			: LREAL;
END_VAR

METHOD Halt : E_CommandResult
ExecuteCommand(INDEX_COMMAND_HALT);

// IF iCommands[INDEX_COMMAND_HALT].P_CommandStatus.Result = E_CommandResult.Accepted THEN
// END_IF
END_METHOD

METHOD MoveRelative : E_CommandResult
VAR_INPUT
	lrDistance	: LREAL := 0.0;
	lrVelocity	: LREAL := AxisConfiguration.lrScrollVelocity;
END_VAR
lrRelDistance := lrDistance;
lrRelVelocity := lrVelocity;
ExecuteCommand(INDEX_COMMAND_MOVERELATIVE);

// IF iCommands[INDEX_COMMAND_MOVERELATIVE] <> 0 THEN
// 	IF iCommands[INDEX_COMMAND_MOVERELATIVE].P_CommandStatus.Result = E_CommandResult.Accepted THEN
// 		lrRelDistance := lrDistance;
// 		lrRelVelocity := lrVelocity;
// 		//bRelativeFlag := TRUE;
// 	END_IF
// ELSE
// 	//TraceWithSeverity()
// END_IF
END_METHOD

METHOD MoveVelocity : E_CommandResult
VAR_INPUT
	lrVelocity	: LREAL := 0.0;
	eDirection	: MC_Direction := MC_Positive_Direction;
END_VAR
lrVelVelocity := lrVelocity;
eVelDirection := eDirection;
ExecuteCommand(INDEX_COMMAND_MOVEVELOCITY);

// IF iCommands[INDEX_COMMAND_MOVEVELOCITY].P_CommandStatus.Result = E_CommandResult.Accepted THEN
// 	lrVelVelocity := lrVelocity;
// 	eVelDirection := eDirection;
// 	//bVelocityFlag := TRUE;
// END_IF
END_METHOD

METHOD PowerOff : E_CommandResult
ExecuteCommand(INDEX_COMMAND_POWEROFF);

IF iCommands[INDEX_COMMAND_POWEROFF].P_CommandStatus.Result = E_CommandResult.Accepted THEN
	bPowerOn := FALSE;
END_IF
END_METHOD

METHOD PowerOn : E_CommandResult
ExecuteCommand(INDEX_COMMAND_POWERON);

IF iCommands[INDEX_COMMAND_POWERON].P_CommandStatus.Result = E_CommandResult.Accepted THEN
	bPowerOn := TRUE;
END_IF
END_METHOD

METHOD ResetAxis : E_CommandResult
ExecuteCommand(INDEX_COMMAND_RESETAXIS);

// IF iCommands[INDEX_COMMAND_RESETAXIS].P_CommandStatus.Result = E_CommandResult.Accepted THEN
// 	bResetFlag := TRUE;
// END_IF
END_METHOD

METHOD SetBrake : E_CommandResult
VAR_INPUT
	eBrakeMode	: Tc2_MC2_Drive.E_BrakeMode := .E_BrakeMode.eBrakeMode_Automatic;
END_VAR
eAxisBrakeMode := eBrakeMode;
ExecuteCommand(INDEX_COMMAND_SETBRAKE);

// IF iCommands[INDEX_COMMAND_SETBRAKE].P_CommandStatus.Result = E_CommandResult.Accepted THEN
// 	eAxisBrakeMode := eBrakeMode;
// 	//bBrakeControlFlag := TRUE;
// END_IF
END_METHOD

METHOD SetTension : E_CommandResult
VAR_INPUT
	lrTorque : LREAL := 0.0; // In Tensies
END_VAR
ExecuteCommand(INDEX_COMMAND_SETTENSION);

IF iCommands[INDEX_COMMAND_SETTENSION].P_CommandStatus.Result = E_CommandResult.Accepted THEN
	lrTorqueTensies	 := lrTorque;	
	bTorqueFlag := TRUE;	
END_IF
END_METHOD

METHOD Stop : E_CommandResult
ExecuteCommand(INDEX_COMMAND_STOP);

Stop := iCommands[INDEX_COMMAND_STOP].P_CommandStatus.Result;
// IF iCommands[INDEX_COMMAND_STOP].P_CommandStatus.Result = E_CommandResult.Accepted THEN
// 	bStopFlag := TRUE;
// END_IF
END_METHOD

METHOD PROTECTED _InitializeReferences : BOOL
//Initialize data references
SUPER^._InitializeReferences();

ComponentConfiguration.BaseConfiguration 			REF= SUPER^.BaseConfiguration;
                                                    
ComponentStatus.BaseStatus							REF= SUPER^.BaseStatus;

ComponentStatus.AmsNetId							REF= ComponentConfiguration.AmsNetId;

AxisConfiguration.ComponentConfiguration			REF= SUPER^.ComponentConfiguration;

AxisStatus.BaseComponentStatus						REF= SUPER^.ComponentStatus;

_InitializeReferences 								:= TRUE; // apply at end of all reference initialization
END_METHOD

METHOD PROTECTED _SetCommandPermIntlkConfiguration : BOOL
CommandPermIntlkConfiguration[INDEX_COMMAND_HALT].P_CommandConfiguration.CommandDescription	:= 'Halt Axis';
CommandPermIntlkConfiguration[INDEX_COMMAND_HALT].P_CommandConfiguration.CommandIndex	:= INDEX_COMMAND_HALT;
CommandPermIntlkConfiguration[INDEX_COMMAND_HALT].P_CommandConfiguration.CommandPOUName	:= 'Halt';
CommandPermIntlkConfiguration[INDEX_COMMAND_HALT].P_CommandConfiguration.CompletionCondition REF= SUPER^.CommandCompletionConditions[INDEX_COMMAND_HALT];

CommandPermIntlkConfiguration[INDEX_COMMAND_MOVERELATIVE].P_CommandConfiguration.CommandDescription	:= 'Move axis by relative distance';
CommandPermIntlkConfiguration[INDEX_COMMAND_MOVERELATIVE].P_CommandConfiguration.CommandIndex	:= INDEX_COMMAND_MOVERELATIVE;
CommandPermIntlkConfiguration[INDEX_COMMAND_MOVERELATIVE].P_CommandConfiguration.CommandPOUName	:= 'MoveRelative';
CommandPermIntlkConfiguration[INDEX_COMMAND_MOVERELATIVE].P_CommandConfiguration.CompletionCondition REF= SUPER^.CommandCompletionConditions[INDEX_COMMAND_MOVERELATIVE];

CommandPermIntlkConfiguration[INDEX_COMMAND_MoveVelocity].P_CommandConfiguration.CommandDescription	:= 'Move axis with given velocity';
CommandPermIntlkConfiguration[INDEX_COMMAND_MoveVelocity].P_CommandConfiguration.CommandIndex	:= INDEX_COMMAND_MOVEVELOCITY;
CommandPermIntlkConfiguration[INDEX_COMMAND_MoveVelocity].P_CommandConfiguration.CommandPOUName	:= 'MoveVelocity';
CommandPermIntlkConfiguration[INDEX_COMMAND_MoveVelocity].P_CommandConfiguration.CompletionCondition REF= SUPER^.CommandCompletionConditions[INDEX_COMMAND_MOVEVELOCITY];

CommandPermIntlkConfiguration[INDEX_COMMAND_POWEROFF].P_CommandConfiguration.CommandDescription	:= 'Power off the axis';
CommandPermIntlkConfiguration[INDEX_COMMAND_POWEROFF].P_CommandConfiguration.CommandIndex	:= INDEX_COMMAND_POWEROFF;
CommandPermIntlkConfiguration[INDEX_COMMAND_POWEROFF].P_CommandConfiguration.CommandPOUName	:= 'PowerOff';
CommandPermIntlkConfiguration[INDEX_COMMAND_POWEROFF].P_CommandConfiguration.CompletionCondition REF= SUPER^.CommandCompletionConditions[INDEX_COMMAND_POWEROFF];

CommandPermIntlkConfiguration[INDEX_COMMAND_POWERON].P_CommandConfiguration.CommandDescription	:= 'Power on the axis';
CommandPermIntlkConfiguration[INDEX_COMMAND_POWERON].P_CommandConfiguration.CommandIndex	:= INDEX_COMMAND_POWERON;
CommandPermIntlkConfiguration[INDEX_COMMAND_POWERON].P_CommandConfiguration.CommandPOUName	:= 'PowerOn';
CommandPermIntlkConfiguration[INDEX_COMMAND_POWERON].P_CommandConfiguration.CompletionCondition REF= SUPER^.CommandCompletionConditions[INDEX_COMMAND_POWERON];

CommandPermIntlkConfiguration[INDEX_COMMAND_RESETAXIS].P_CommandConfiguration.CommandDescription	:= 'Reset axis errors';
CommandPermIntlkConfiguration[INDEX_COMMAND_RESETAXIS].P_CommandConfiguration.CommandIndex	:= INDEX_COMMAND_RESETAXIS;
CommandPermIntlkConfiguration[INDEX_COMMAND_RESETAXIS].P_CommandConfiguration.CommandPOUName	:= 'ResetAxis';
CommandPermIntlkConfiguration[INDEX_COMMAND_RESETAXIS].P_CommandConfiguration.CompletionCondition REF= SUPER^.CommandCompletionConditions[INDEX_COMMAND_RESETAXIS];

CommandPermIntlkConfiguration[INDEX_COMMAND_SETBRAKE].P_CommandConfiguration.CommandDescription	:= 'Set brake mode of the axis.';
CommandPermIntlkConfiguration[INDEX_COMMAND_SETBRAKE].P_CommandConfiguration.CommandIndex	:= INDEX_COMMAND_SETBRAKE;
CommandPermIntlkConfiguration[INDEX_COMMAND_SETBRAKE].P_CommandConfiguration.CommandPOUName	:= 'SetBrake';
CommandPermIntlkConfiguration[INDEX_COMMAND_SETBRAKE].P_CommandConfiguration.CompletionCondition REF= SUPER^.CommandCompletionConditions[INDEX_COMMAND_SETBRAKE];

CommandPermIntlkConfiguration[INDEX_COMMAND_SETTENSION].P_CommandConfiguration.CommandDescription	:= 'Set tensies on torque block.';
CommandPermIntlkConfiguration[INDEX_COMMAND_SETTENSION].P_CommandConfiguration.CommandIndex	:= INDEX_COMMAND_SETTENSION;
CommandPermIntlkConfiguration[INDEX_COMMAND_SETTENSION].P_CommandConfiguration.CommandPOUName	:= 'SetTension';
CommandPermIntlkConfiguration[INDEX_COMMAND_SETTENSION].P_CommandConfiguration.CompletionCondition REF= SUPER^.CommandCompletionConditions[INDEX_COMMAND_SETTENSION];

CommandPermIntlkConfiguration[INDEX_COMMAND_STOP].P_CommandConfiguration.CommandDescription	:= 'Uninterruptable stop of the axis.';
CommandPermIntlkConfiguration[INDEX_COMMAND_STOP].P_CommandConfiguration.CommandIndex	:= INDEX_COMMAND_STOP;
CommandPermIntlkConfiguration[INDEX_COMMAND_STOP].P_CommandConfiguration.CommandPOUName	:= 'Stop';
CommandPermIntlkConfiguration[INDEX_COMMAND_STOP].P_CommandConfiguration.CompletionCondition REF= SUPER^.CommandCompletionConditions[INDEX_COMMAND_STOP];

_SetCommandPermIntlkConfiguration	:= TRUE;
END_METHOD

METHOD PROTECTED _BeckhoffMotionFBs
fbPower(
	Axis:= Axis, 
	Enable:= bPowerOn, 
	Enable_Positive:= bPowerOn, 
	Enable_Negative:= bPowerOn, 
	Override:= lrOverridePower);

fbReset(
	Axis:= Axis, 
	Execute:= bResetFlag);
	
fbHalt(
	Axis:= Axis, 
	Execute:= bHaltFlag);
	
fbRelative(
	Axis:= Axis, 
	Execute:= bRelativeFlag, 
	Distance:= lrRelDistance, 
	Velocity:= lrRelVelocity);
	
fbVelocity(
	Axis:= Axis, 
	Execute:= bVelocityFlag, 
	Velocity:= lrVelVelocity,
	Direction:= eVelDirection);
	
fbTorque(
	Axis:= Axis, 
	Execute:= bTorqueFlag, 
	ContinuousUpdate:= TRUE, 
	Relative:= FALSE, 
	Torque:= lrTorqueTensies, 
	TorqueRamp:= AxisConfiguration.lrTorqueRamp, 
	VelocityLimitHigh:= AxisConfiguration.lrMaxSpeed, 
	VelocityLimitLow:= -AxisConfiguration.lrMaxSpeed);
	
fbStop(
	Axis:= Axis,
	Execute:= bStopFlag);

fbBrakeControl(
	Axis:= Axis, 
	Execute:= bBrakeControlFlag, 
	Mode:= eAxisBrakeMode);
END_METHOD

METHOD PROTECTED _CyclicFlags
// Base implementation - Component derivatives should override this method
// This method maps from command index to business logic method calls
bHaltFlag := iCommands[INDEX_COMMAND_HALT].P_CommandStatus.BaseStatus.Busy;
bRelativeFlag := iCommands[INDEX_COMMAND_MOVERELATIVE].P_CommandStatus.BaseStatus.Busy;
bVelocityFlag := iCommands[INDEX_COMMAND_MOVEVELOCITY].P_CommandStatus.BaseStatus.Busy;
bResetFlag := iCommands[INDEX_COMMAND_RESETAXIS].P_CommandStatus.BaseStatus.Busy;
bBrakeControlFlag := iCommands[INDEX_COMMAND_SETBRAKE].P_CommandStatus.BaseStatus.Busy;
bStopFlag := iCommands[INDEX_COMMAND_STOP].P_CommandStatus.BaseStatus.Busy;



	// Invalid index - trace error
IF SUPER^.BaseConfiguration.LogTraceConfiguration.What.xLogToEventLogger THEN
	TraceWithSeverity(Message := 'Invalid CommandIndex in _ExecuteCommandByIndex', Severity := Global.TcEventSeverity.Warning);
END_IF
END_METHOD

(*
Example Implementation:
// Set completion conditions - commands complete immediately after transitioning to acting state
// This prevents the component from staying busy and blocking other commands
SUPER^.CommandCompletionConditions[INDEX_COMMAND_ABORT]            		:= (SequencerStatus.CurrentState = E_PackMLState.Aborting);
SUPER^.CommandCompletionConditions[INDEX_COMMAND_CLEAR]            		:= (SequencerStatus.CurrentState = E_PackMLState.Clearing);
SUPER^.CommandCompletionConditions[INDEX_COMMAND_COMPLETE]         		:= (SequencerStatus.CurrentState = E_PackMLState.Completing);
SUPER^.CommandCompletionConditions[INDEX_COMMAND_HOLD]             		:= (SequencerStatus.CurrentState = E_PackMLState.Holding);
SUPER^.CommandCompletionConditions[INDEX_COMMAND_RESET]            		:= (SequencerStatus.CurrentState = E_PackMLState.Resetting);
SUPER^.CommandCompletionConditions[INDEX_COMMAND_RESUMEFROMHOLD]   		:= (SequencerStatus.CurrentState = E_PackMLState.Unholding);
SUPER^.CommandCompletionConditions[INDEX_COMMAND_RESUMEFROMSUSPEND]		:= (SequencerStatus.CurrentState = E_PackMLState.Unsuspending);
SUPER^.CommandCompletionConditions[INDEX_COMMAND_START]            		:= (SequencerStatus.CurrentState = E_PackMLState.Starting);
SUPER^.CommandCompletionConditions[INDEX_COMMAND_STOP]             		:= (SequencerStatus.CurrentState = E_PackMLState.Stopping);
SUPER^.CommandCompletionConditions[INDEX_COMMAND_SUSPEND]          		:= (SequencerStatus.CurrentState = E_PackMLState.Suspending);

// Enable/Disable don't have specific PackML states, handle as needed
SUPER^.CommandCompletionConditions[INDEX_COMMAND_ENABLE]           		:= (NOT SUPER^.BaseStatus.Enabled);
SUPER^.CommandCompletionConditions[INDEX_COMMAND_DISABLE]          		:= SUPER^.BaseStatus.Enabled;

_EvaluateCompletionConditions	:= TRUE;
*)
METHOD PROTECTED _EvaluateCompletionConditions : BOOL
SUPER^.CommandCompletionConditions[INDEX_COMMAND_HALT]       	 		:= fbHalt.Done;
SUPER^.CommandCompletionConditions[INDEX_COMMAND_MOVERELATIVE]      	:= fbRelative.Done;
SUPER^.CommandCompletionConditions[INDEX_COMMAND_MOVEVELOCITY]       	:= fbVelocity.InVelocity;
SUPER^.CommandCompletionConditions[INDEX_COMMAND_POWEROFF]      		:= NOT fbPower.Status AND NOT fbPower.Busy;
SUPER^.CommandCompletionConditions[INDEX_COMMAND_POWERON]      			:= fbPower.Status AND fbPower.Busy;
SUPER^.CommandCompletionConditions[INDEX_COMMAND_RESETAXIS]      		:= fbReset.Done;
SUPER^.CommandCompletionConditions[INDEX_COMMAND_SETBRAKE]      		:= NOT fbBrakeControl.Busy;
SUPER^.CommandCompletionConditions[INDEX_COMMAND_SETTENSION]      		:= fbTorque.InTorque;
SUPER^.CommandCompletionConditions[INDEX_COMMAND_STOP]      			:= fbStop.Done;



_EvaluateCompletionConditions	:= TRUE;
END_METHOD

(* Example implementation from FB_Actuator:
IF ActuatorStatus.ExtendOutput AND NOT ActuatorStatus.RetractOutput THEN
	ActuatorStatus.ActuatorState	:= E_ActuatorState.Extended;
ELSIF ActuatorStatus.RetractOutput AND NOT ActuatorStatus.ExtendOutput THEN
	ActuatorStatus.ActuatorState	:= E_ActuatorState.Retracted;
ELSE
	ActuatorStatus.ActuatorState	:= E_ActuatorState.Indeterminate;
END_IF

_UpdateComponentStatus := THIS^;*)
METHOD PROTECTED _UpdateComponentStatus : Base.I_ComponentFull
END_METHOD

PROPERTY Busy : BOOL
GET
IF __ISVALIDREF(SUPER^.ComponentStatus.BaseStatus) THEN
	Busy := bAxisBusy OR SUPER^.ComponentStatus.BaseStatus.Busy;
ELSE
	Busy := bAxisBusy;
END_IF
END_GET
END_PROPERTY

PROPERTY PUBLIC P_AxisConfiguration : REFERENCE TO ST_BeckhoffAxisConfiguration
GET
P_AxisConfiguration REF= AxisConfiguration;
END_GET
END_PROPERTY

PROPERTY PUBLIC P_AxisReference : REFERENCE TO AXIS_REF
GET
P_AxisReference REF= Axis;
END_GET
END_PROPERTY

PROPERTY P_InTension : BOOL
GET
P_InTension := fbTorque.InTorque;
END_GET
END_PROPERTY

PROPERTY P_Powered : BOOL
GET
P_Powered := bPowered;
END_GET
END_PROPERTY

PROPERTY P_RotaryAxisStatus : REFERENCE TO ST_BeckhoffAxisStatus
GET
P_RotaryAxisStatus REF= AxisStatus;
END_GET
END_PROPERTY

METHOD CyclicLogic

VAR
END_VAR
SUPER^.CyclicLogic();
		
bPowered := fbPower.Status;
bAxisBusy := fbStop.Busy OR fbVelocity.Busy OR fbRelative.Busy OR fbHalt.Busy OR fbBrakeControl.Busy OR fbStop.Busy;
AxisStatus.BaseComponentStatus.BaseStatus.Error := fbPower.Error OR fbTorque.Error OR fbStop.Error OR fbVelocity.Error OR fbRelative.Error OR fbHalt.Error OR fbBrakeControl.Error OR fbStop.Error;

IF AxisStatus.BaseComponentStatus.BaseStatus.Error THEN
	IF fbPower.Error THEN
		AxisStatus.BaseComponentStatus.BaseStatus.ErrorID := fbPower.ErrorId;
	ELSIF fbStop.Error THEN
		AxisStatus.BaseComponentStatus.BaseStatus.ErrorID := fbStop.ErrorId;
	ELSIF fbHalt.Error THEN
		AxisStatus.BaseComponentStatus.BaseStatus.ErrorID := fbHalt.ErrorId;
	ELSIF fbRelative.Error THEN
		AxisStatus.BaseComponentStatus.BaseStatus.ErrorID := fbRelative.ErrorId;
	ELSIF fbVelocity.Error THEN
		AxisStatus.BaseComponentStatus.BaseStatus.ErrorID := fbVelocity.ErrorId;
	ELSIF fbReset.Error THEN
		AxisStatus.BaseComponentStatus.BaseStatus.ErrorID := fbReset.ErrorId;
	ELSIF fbBrakeControl.Error THEN
		AxisStatus.BaseComponentStatus.BaseStatus.ErrorID := fbBrakeControl.ErrorId;
	ELSIF fbTorque.Error THEN
		AxisStatus.BaseComponentStatus.BaseStatus.ErrorID := fbTorque.ErrorId;
// 	ELSE
// 		Trace("Unknown source of error!");
	END_IF
END_IF

_CyclicFlags();
_BeckhoffMotionFBs();
END_METHOD

END_FUNCTION_BLOCK

// ITFs/Motion/I_RotaryAxis
INTERFACE I_RotaryAxis EXTENDS I_BaseCyclic

PROPERTY PUBLIC P_AxisReference : REFERENCE TO AXIS_REF
GET
END_GET
END_PROPERTY

PROPERTY P_RotaryAxisStatus : REFERENCE TO ST_BeckhoffAxisStatus
GET
END_GET
END_PROPERTY

METHOD Halt : Base.E_CommandResult
VAR_INPUT
END_VAR
END_METHOD

METHOD MoveRelative : Base.E_CommandResult
VAR_INPUT
	lrDistance : LREAL := 0.0;
	lrVelocity : LREAL := 0.0;
END_VAR
END_METHOD

METHOD MoveVelocity : Base.E_CommandResult
VAR_INPUT
	lrVelocity	: LREAL := 0.0;
	eDirection 	: MC_Direction := MC_Positive_Direction;
END_VAR
END_METHOD

METHOD PowerOff : Base.E_CommandResult
VAR_INPUT
END_VAR
END_METHOD

METHOD PowerOn : Base.E_CommandResult
VAR_INPUT
END_VAR
END_METHOD

METHOD ResetAxis : Base.E_CommandResult
VAR_INPUT
END_VAR
END_METHOD

METHOD SetBrake : Base.E_CommandResult
VAR_INPUT
	eBrakeMode 		: Tc2_MC2_Drive.E_BrakeMode := E_BrakeMode.eBrakeMode_Automatic;
END_VAR
END_METHOD

METHOD SetTension : Base.E_CommandResult
VAR_INPUT
	lrTorque : LREAL := 0.0; // In Tensies
END_VAR
END_METHOD

METHOD Stop : Base.E_CommandResult
VAR_INPUT
END_VAR
END_METHOD

END_INTERFACE

// BeckhoffAxis/POUs/FB_WebDrive
FUNCTION_BLOCK FB_WebDrive EXTENDS FB_BaseCyclic
VAR
	// Child components
	Tensioner	: FB_BeckhoffAxis;
	Winder		: FB_BeckhoffAxis;
	Encoder		: FB_RotaryEncoder;
	
	bError : BOOL;
	udErrorCode : UDINT;
	
	eState : E_WebDriveState := E_WebDriveState.INIT;
	
	// HMI Set Values
	lrTensionSet  : LREAL := 0.0; // in real Tension
	lrScrollDist  : LREAL := 0.0; // in mm
	
	// Button watchers
	fbScrollTrigger   : R_TRIG;
	fbTensionTrigger  : R_TRIG;
	fbCalibrationTrigger : R_TRIG;
	
	// Encoder Distance Reading
	lrDistanceTraveled : LREAL := 0.0;
	
	// Roll-Radius Scaling
	lrScrollScaleFactor : LREAL := 1.0;
	
	lrWinderAngleTurned : LREAL := 0.0;
	lrWinderRollRadius : LREAL := 60.0; // mm
	lrWinderlastAngle  : LREAL := 0.0;
	
	lrTensionerAngleTurned : LREAL := 0.0;
	lrTensionerRollRadius : LREAL := 60.0; // mm
	lrTensionerlastAngle  : LREAL := 0.0;
	
	// HMI Button Placeholders
	bScrollButton : BOOL;
	bTensionButton : BOOL;
	bCalibrationButton : BOOL;
	
	// Are our current radii accurate?
	bCalibrated : BOOL := FALSE;
END_VAR

METHOD PROTECTED _CalculateRadius : BOOL
VAR_INPUT
END_VAR
lrDistanceTraveled := Encoder.Read();

lrWinderAngleTurned := Winder.P_AxisReference.NcToPlc.ModuloActPos - lrWinderlastAngle;
lrTensionerAngleTurned := Tensioner.P_AxisReference.NcToPlc.ModuloActPos - lrTensionerlastAngle;

IF lrWinderAngleTurned > 1800 THEN
	lrWinderAngleTurned := lrWinderAngleTurned - 3600;
ELSIF lrWinderAngleTurned < -1800 THEN
	lrWinderAngleTurned := lrWinderAngleTurned + 3600;
END_IF

IF lrTensionerAngleTurned > 1800 THEN
	lrTensionerAngleTurned := lrTensionerAngleTurned - 3600;
ELSIF lrTensionerAngleTurned < -1800 THEN
	lrTensionerAngleTurned := lrTensionerAngleTurned + 3600;
END_IF
	
lrWinderRollRadius := (lrDistanceTraveled*3600.0)/(ABS(lrWinderAngleTurned) * 2*pi);
lrTensionerRollRadius := (lrDistanceTraveled*3600.0)/(ABS(lrTensionerAngleTurned) * 2*pi);

lrScrollScaleFactor := 3600.0/(2*pi*lrWinderRollRadius);

lrWinderlastAngle := Winder.P_AxisReference.NcToPlc.ModuloActPos;
lrTensionerlastAngle := Tensioner.P_AxisReference.NcToPlc.ModuloActPos;

bCalibrated := TRUE;
END_METHOD

METHOD PROTECTED _InitializeChildrenDependencies : BOOL
Tensioner.Initialize();
Winder.Initialize();
Encoder.Initialize();

_InitializeChildrenDependencies := TRUE;
END_METHOD

METHOD CyclicLogic
// Call child cyclics
Tensioner.CyclicLogic();
Winder.CyclicLogic();
Encoder.CyclicLogic();

// Check for web errors
IF Tensioner.Error OR Winder.Error THEN
	eState := E_WebDriveState.ERROR;
	
	IF Tensioner.Error THEN
		udErrorCode := Tensioner.ErrorID;
	ELSIF Winder.Error THEN
		udErrorCode := Winder.ErrorID; 
	END_IF
END_IF


CASE eState OF
	E_WebDriveState.INIT:
		Tensioner.PowerOn();
		Winder.PowerOn();
		IF Tensioner.P_Powered AND Winder.P_Powered THEN
			Tensioner.SetTension(0.0); // idle tension
			Winder.Halt(); // Ensure winder is not moving
			
			// Initialize Readings
			lrWinderlastAngle := Winder.P_AxisReference.NcToPlc.ModuloActPos;
			lrTensionerlastAngle := Tensioner.P_AxisReference.NcToPlc.ModuloActPos;
			Encoder.Read();
			
			eState := E_WebDriveState.IDLE;
		END_IF
	E_WebDriveState.CALIBRATION:
		IF NOT Tensioner.Busy THEN
			Winder.MoveRelative(-50.0, Winder.P_AxisConfiguration.lrScrollVelocity);
			eState := E_WebDriveState.BUSY_SCROLL;
		END_IF
	E_WebDriveState.IDLE:
		IF fbScrollTrigger.Q THEN
			Winder.MoveRelative(-lrScrollDist*lrScrollScaleFactor, Winder.P_AxisConfiguration.lrScrollVelocity);
			eState := E_WebDriveState.BUSY_SCROLL;
		ELSIF fbTensionTrigger.Q THEN
			Tensioner.SetTension(((lrTensionSet*lrTensionerRollRadius/1000) - 1.0748)/0.5314); // conversion from Tension to tensies
			eState := E_WebDriveState.BUSY_TENSION;
		ELSIF fbCalibrationTrigger.Q THEN
			Tensioner.SetTension(50.0); // Calibration tension, 50
			eState := E_WebDriveState.CALIBRATION;
		ELSIF Encoder.Read() > 0.1 THEN
			eState := E_WebDriveState.ERROR;
		END_IF
		
		
	E_WebDriveState.BUSY_TENSION:
		IF NOT Tensioner.Busy THEN
			Encoder.Read(); // get rid of any slight skip that happened as a result of applying tension
			eState := E_WebDriveState.IDLE;
		END_IF
		
		
	E_WebDriveState.BUSY_SCROLL:
		IF NOT Winder.Busy THEN
			_CalculateRadius();
			eState := E_WebDriveState.IDLE;
		END_IF
		
		
	E_WebDriveState.ERROR:
		Tensioner.Stop();
		Winder.Stop();
END_CASE

// Watch for HMI button presses
fbScrollTrigger(CLK:= bScrollButton, Q=>);
fbTensionTrigger(CLK:= bTensionButton, Q=>);
fbCalibrationTrigger(CLK:= bCalibrationButton, Q=>);
END_METHOD

END_FUNCTION_BLOCK

// RotaryEncoder/POUs/FB_RotaryEncoder
FUNCTION_BLOCK FB_RotaryEncoder EXTENDS FB_Component<GC_RotaryEncoder.INDEX_COMMAND_MIN,GC_RotaryEncoder.INDEX_COMMAND_MAX> IMPLEMENTS I_RotaryEncoder

VAR CONSTANT
	INDEX_COMMAND_READ : DINT := 0;
END_VAR


VAR
	EncoderConfiguration 	: ST_RotaryEncoderConfiguration;
	EncoderStatus			: ST_RotaryEncoderStatus;
	encoderValue AT %I* : UINT;
	
	lastValue : UINT := 0;
	diff 	  : DINT := 0;
END_VAR

METHOD Read : LREAL
ExecuteCommand(INDEX_COMMAND_READ);

IF iCommands[INDEX_COMMAND_READ].P_CommandStatus.Result = E_CommandResult.Accepted THEN
	diff := encoderValue - lastValue;
	IF diff > 32768 THEN
		diff := diff - 65536;
	ELSIF diff < -32768 THEN
		diff := diff + 65536;
	END_IF
	
	IF EncoderConfiguration.CPmm <> 0 THEN
		Read := DINT_TO_LREAL(diff)/EncoderConfiguration.CPmm;
	END_IF
	
	lastValue := encoderValue;
END_IF
END_METHOD

METHOD PROTECTED _InitializeReferences : BOOL
//Initialize data references
SUPER^._InitializeReferences();

ComponentConfiguration.BaseConfiguration 			REF= SUPER^.BaseConfiguration;
                                                    
ComponentStatus.BaseStatus							REF= SUPER^.BaseStatus;

ComponentStatus.AmsNetId							REF= ComponentConfiguration.AmsNetId;

EncoderConfiguration.ComponentConfiguration			REF= SUPER^.ComponentConfiguration;

EncoderStatus.BaseComponentStatus						REF= SUPER^.ComponentStatus;

_InitializeReferences 								:= TRUE; // apply at end of all reference initialization
END_METHOD

METHOD PROTECTED _SetCommandPermIntlkConfiguration : BOOL
CommandPermIntlkConfiguration[INDEX_COMMAND_READ].P_CommandConfiguration.CommandDescription	:= 'Read the distance travelled on the encoder since the last read.';
CommandPermIntlkConfiguration[INDEX_COMMAND_READ].P_CommandConfiguration.CommandIndex	:= INDEX_COMMAND_READ;
CommandPermIntlkConfiguration[INDEX_COMMAND_READ].P_CommandConfiguration.CommandPOUName	:= 'Read';
CommandPermIntlkConfiguration[INDEX_COMMAND_READ].P_CommandConfiguration.CompletionCondition REF= SUPER^.CommandCompletionConditions[INDEX_COMMAND_READ];

_SetCommandPermIntlkConfiguration	:= TRUE;
END_METHOD

(*
Example Implementation:
// Set completion conditions - commands complete immediately after transitioning to acting state
// This prevents the component from staying busy and blocking other commands
SUPER^.CommandCompletionConditions[INDEX_COMMAND_ABORT]            		:= (SequencerStatus.CurrentState = E_PackMLState.Aborting);
SUPER^.CommandCompletionConditions[INDEX_COMMAND_CLEAR]            		:= (SequencerStatus.CurrentState = E_PackMLState.Clearing);
SUPER^.CommandCompletionConditions[INDEX_COMMAND_COMPLETE]         		:= (SequencerStatus.CurrentState = E_PackMLState.Completing);
SUPER^.CommandCompletionConditions[INDEX_COMMAND_HOLD]             		:= (SequencerStatus.CurrentState = E_PackMLState.Holding);
SUPER^.CommandCompletionConditions[INDEX_COMMAND_RESET]            		:= (SequencerStatus.CurrentState = E_PackMLState.Resetting);
SUPER^.CommandCompletionConditions[INDEX_COMMAND_RESUMEFROMHOLD]   		:= (SequencerStatus.CurrentState = E_PackMLState.Unholding);
SUPER^.CommandCompletionConditions[INDEX_COMMAND_RESUMEFROMSUSPEND]		:= (SequencerStatus.CurrentState = E_PackMLState.Unsuspending);
SUPER^.CommandCompletionConditions[INDEX_COMMAND_START]            		:= (SequencerStatus.CurrentState = E_PackMLState.Starting);
SUPER^.CommandCompletionConditions[INDEX_COMMAND_STOP]             		:= (SequencerStatus.CurrentState = E_PackMLState.Stopping);
SUPER^.CommandCompletionConditions[INDEX_COMMAND_SUSPEND]          		:= (SequencerStatus.CurrentState = E_PackMLState.Suspending);

// Enable/Disable don't have specific PackML states, handle as needed
SUPER^.CommandCompletionConditions[INDEX_COMMAND_ENABLE]           		:= (NOT SUPER^.BaseStatus.Enabled);
SUPER^.CommandCompletionConditions[INDEX_COMMAND_DISABLE]          		:= SUPER^.BaseStatus.Enabled;

_EvaluateCompletionConditions	:= TRUE;
*)
METHOD PROTECTED _EvaluateCompletionConditions : BOOL
SUPER^.CommandCompletionConditions[INDEX_COMMAND_READ]       	 		:= lastValue = encoderValue;



_EvaluateCompletionConditions	:= TRUE;
END_METHOD

(* Example implementation from FB_Actuator:
IF ActuatorStatus.ExtendOutput AND NOT ActuatorStatus.RetractOutput THEN
	ActuatorStatus.ActuatorState	:= E_ActuatorState.Extended;
ELSIF ActuatorStatus.RetractOutput AND NOT ActuatorStatus.ExtendOutput THEN
	ActuatorStatus.ActuatorState	:= E_ActuatorState.Retracted;
ELSE
	ActuatorStatus.ActuatorState	:= E_ActuatorState.Indeterminate;
END_IF

_UpdateComponentStatus := THIS^;*)
METHOD PROTECTED _UpdateComponentStatus : Base.I_ComponentFull
END_METHOD

METHOD CyclicLogic
SUPER^.CyclicLogic();
END_METHOD

END_FUNCTION_BLOCK

// ITFs/Motion/I_RotaryEncoder
INTERFACE I_RotaryEncoder EXTENDS I_BaseCyclic

METHOD Read : LREAL
VAR_INPUT
END_VAR
END_METHOD

END_INTERFACE

// ITFs/Motion/I_CompleteAxis
INTERFACE I_CompleteAxis EXTENDS I_RotaryAxis

METHOD MoveAbsolute : Base.E_CommandResult
VAR_INPUT
END_VAR
END_METHOD

END_INTERFACE

// Zaber/POUs/Functions/F_ExtractAxisNumber
FUNCTION F_ExtractAxisNumber : STRING
VAR_INPUT  sInput : STRING;  END_VAR
VAR
    Tok : ARRAY[1..16] OF STRING;
    i   : INT;
END_VAR

Tok := F_ZaberSplitReplyTokensEx(sInput := sInput);

IF Tok[2] <> '' THEN
    F_ExtractAxisNumber := Tok[2];
ELSE
    F_ExtractAxisNumber := '';
END_IF

END_FUNCTION

// Zaber/POUs/Functions/F_ZaberSplitReplyTokensEx
(*
======================================================================
  F_SplitReplyTokensEx  (FOR-only version)
  • Splits a Zaber reply into ≤16 tokens.
  • Uses only bounded FOR loops.
  • Returns ARRAY[1..16] OF STRING (unused slots = '').
======================================================================
*)
FUNCTION F_ZaberSplitReplyTokensEx : ARRAY[1..16] OF STRING
VAR_INPUT
    sInput : STRING;
END_VAR
VAR
    Tok       : ARRAY[1..16] OF STRING;
    work      : STRING;
    i, k      : INT;
    posSpace  : INT;
    leading   : INT;
END_VAR

(* ---------- clear output array ---------------------------- *)
FOR i := 1 TO 16 DO
	Tok[i] := '';
END_FOR

(* ---------- trim trailing CR / LF ------------------------- *)
work := sInput;
FOR i := LEN(work) TO 1 BY -1 DO
	IF (MID(work,i,1) <> Tc2_System.F_ToCHR(13)) AND (MID(work,i,1) <> Tc2_System.F_ToCHR(10)) THEN
		work := LEFT(work,i);
		EXIT;                       (* done trimming *)
	END_IF
END_FOR

(* ---------- tokenise  (max 16 loops) ---------------------- *)
FOR i := 1 TO 16 DO
	IF work = '' THEN EXIT; END_IF     (* nothing left *)

	(* 1) skip leading spaces with bounded scan *)
	leading := 0;
	FOR k := 1 TO LEN(work) DO
		IF MID(work,k,1) = ' ' THEN
			leading := leading + 1;
		ELSE
			EXIT;   (* first non-space found *)
		END_IF
	END_FOR
	IF leading > 0 THEN
		work := RIGHT(work, LEN(work) - leading);
		IF work = '' THEN EXIT; END_IF
	END_IF

	(* 2) locate next space *)
	posSpace := FIND(work, ' ');

	IF posSpace = 0 THEN               (* last token *)
		Tok[i] := work;
		EXIT;                           (* done *)
	ELSE                                (* token before next space *)
		Tok[i] := LEFT(work, posSpace - 1);
		work   := RIGHT(work, LEN(work) - posSpace);
	END_IF
END_FOR

(* ---------- return token array ---------------------------- *)
F_ZaberSplitReplyTokensEx := Tok;

END_FUNCTION

// Zaber/POUs/Functions/F_ExtractDataField
FUNCTION F_ExtractDataField : STRING
VAR_INPUT
    sInput : STRING;
END_VAR
VAR
    Tok         : ARRAY[1..16] OF STRING;
    dataStart   : INT;
    i, d        : INT;
    hasMsgID    : BOOL := FALSE;
    firstChar   : STRING(1);
    piece       : STRING;
    outStr      : STRING := '';
END_VAR

(* 1) Tokenise once *)
Tok := F_ZaberSplitReplyTokensEx(sInput := sInput);

(* 2) Detect 2-digit numeric Message-ID in Tok[3] when Tok[4] is OK/RJ *)
IF (TOK[4] = 'OK') OR (TOK[4] = 'RJ') THEN
    IF LEN(Tok[3]) = 2 THEN
        firstChar := MID(Tok[3],1,1);
        FOR d := 0 TO 9 DO
            IF firstChar = INT_TO_STRING(d) THEN
                hasMsgID := TRUE;
                EXIT;
            END_IF
        END_FOR
    END_IF
END_IF

(* 3) Decide data-start index *)
IF hasMsgID THEN
    dataStart := 7;   (* @nn 0 01 OK BUSY/IDLE --  [data…] *)
ELSE
    dataStart := 6;   (* @nn 0 OK BUSY/IDLE --  [data…]   *)
END_IF

(* 4) Collect tokens until checksum *)
FOR i := dataStart TO 16 DO
    IF Tok[i] = '' THEN
        EXIT;                         (* end of tokens *)
    END_IF

    (* a) Pure checksum token begins with ':' *)
    IF LEFT(Tok[i],1) = ':' THEN
        EXIT;
    END_IF

    (* b) Embedded checksum 'word:CC' *)
    IF FIND(Tok[i], ':') > 0 THEN
        piece := LEFT(Tok[i], FIND(Tok[i], ':') - 1);
        IF piece <> '' THEN
            IF outStr = '' THEN
                outStr := piece;
            ELSE
                outStr := CONCAT(outStr, ' ');
                outStr := CONCAT(outStr, piece);
            END_IF
        END_IF
        EXIT;                         (* checksum reached, stop *)
    END_IF

    (* c) Normal data token *)
    IF outStr = '' THEN
        outStr := Tok[i];
    ELSE
        outStr := CONCAT(outStr, ' ');
        outStr := CONCAT(outStr, Tok[i]);
    END_IF
END_FOR

F_ExtractDataField := outStr;

END_FUNCTION

// Zaber/POUs/Functions/F_ExtractDeviceAddress
(*
======================================================================
  F_ExtractDeviceAddress
======================================================================
*)
FUNCTION F_ExtractDeviceAddress : STRING
VAR_INPUT  sInput : STRING;  END_VAR
VAR
    Tok        : ARRAY[1..16] OF STRING;
    i          : INT;
    deviceAddr : STRING := '';
END_VAR

Tok := F_ZaberSplitReplyTokensEx(sInput := sInput);

IF Tok[1] <> '' THEN
    (* '@01' -> '01' *)
    deviceAddr := RIGHT(Tok[1], LEN(Tok[1]) - 1);
END_IF

F_ExtractDeviceAddress := deviceAddr;

END_FUNCTION

// Zaber/POUs/Functions/F_ExtractMessageChecksum
(*======================================================================
  F_ExtractMessageChecksum
  Returns ":CC" portion (including ':') if present.
======================================================================*)
FUNCTION F_ExtractMessageChecksum : Tc2_System.T_MaxString
VAR_INPUT
    sInput : Tc2_System.T_MaxString;   // Input string
END_VAR
VAR
    i           : INT;
    strLength   : INT;
    bChar       : BYTE := 58;          // ASCII value of ':'  (16#3A)
    resultStr   : Tc2_System.T_MaxString;
    arrInput    : ARRAY[0..255] OF BYTE;
    bFound      : BOOL := FALSE;
END_VAR

strLength := LEN(sInput);
IF strLength = 0 THEN
    F_ExtractMessageChecksum := '';
    RETURN;
END_IF

arrInput := Tc2_Utilities.MAXSTRING_TO_BYTEARR(sInput);  // string → BYTE array

// 1) Check if a ':' exists at all (scan right→left once, stop on first hit)
FOR i := strLength TO 1 BY -1 DO
    IF arrInput[i] = bChar THEN
        bFound := TRUE;
        EXIT;
    END_IF
END_FOR

IF NOT bFound THEN
    // No colon in the string → return empty
    F_ExtractMessageChecksum := '';
    RETURN;
END_IF

// 2) If last character is ':' → nothing after it, return empty
IF arrInput[strLength] = bChar THEN
    F_ExtractMessageChecksum := '';
    RETURN;
END_IF

// 3) Build result by prepending characters right-to-left
resultStr := '';
FOR i := strLength TO 1 BY -1 DO
    IF arrInput[i] = bChar THEN
        EXIT;                         // reached the colon
    END_IF
    resultStr := Tc2_Standard.CONCAT(Tc2_System.F_ToCHR(arrInput[i]), resultStr);
END_FOR

F_ExtractMessageChecksum := resultStr;

END_FUNCTION

// Zaber/POUs/Functions/F_ExtractMotionStatus
FUNCTION F_ExtractMotionStatus : STRING
VAR_INPUT  sInput : STRING;  END_VAR
VAR
    Tok         : ARRAY[1..16] OF STRING;
    i, idx      : INT;
    statusTok   : STRING := '';
END_VAR

Tok := F_ZaberSplitReplyTokensEx(sInput := sInput);

IF (LEN(Tok[3]) = 2) AND (Tok[4] = 'OK' OR Tok[4] = 'RJ') THEN
	idx := 5;  (* ID present *)
ELSE
	idx := 4;
END_IF

statusTok := Tok[idx];
IF (statusTok = 'BUSY') OR (statusTok = 'IDLE') THEN
	F_ExtractMotionStatus := statusTok;
ELSE
	F_ExtractMotionStatus := '';
END_IF

END_FUNCTION

// Zaber/POUs/Functions/F_ZaberExtractExecutionResult
FUNCTION F_ZaberExtractExecutionResult : STRING
VAR_INPUT  sInput : STRING;  END_VAR
VAR
    Tok      : ARRAY[1..16] OF STRING;
    RJ_List  : ARRAY[1..21] OF STRING := [
        'AGAIN','AXISONLY','BADAXIS','BADCOMMAND','BADDATA','BADMESSAGEID',
        'BADSPLIT','DEVICEONLY','DRIVERDISABLED','FULL','INACTIVE','LOCKSTEP',
        'LONGWORD','NOACCESS','NOTSIN','NOTSUPPORTED','PARKED','STATUSBUSY',
        'SYSTEMERROR','TWISTED','OVERDRIVELIMIT'
    ];
    i, idx   : INT;
    baseFlag : STRING := '';
    subcode  : STRING := '';
    okSub    : BOOL  := FALSE;
    outStr   : STRING := '';
END_VAR

Tok := F_ZaberSplitReplyTokensEx(sInput := sInput);

(* decide where the flag sits *)
IF (LEN(Tok[3]) = 2) AND (Tok[4] = 'OK' OR Tok[4] = 'RJ') THEN
    idx := 4;   (* message-ID present *)
ELSE
    idx := 3;
END_IF

baseFlag := Tok[idx];
outStr   := baseFlag;

IF baseFlag = 'RJ' THEN
    subcode := Tok[idx + 1];
    FOR i := 1 TO 21 DO
        IF subcode = RJ_List[i] THEN
            okSub := TRUE;
            EXIT;
        END_IF
    END_FOR
    IF okSub THEN
        outStr := CONCAT(baseFlag, ' ');
        outStr := CONCAT(outStr, subcode);
    END_IF
END_IF

F_ZaberExtractExecutionResult := outStr;

END_FUNCTION

// Zaber/POUs/Functions/F_ZaberExtractWarnFaultFlag
FUNCTION F_ZaberExtractWarnFaultFlag : STRING
VAR_INPUT
    sInput : STRING;
END_VAR
VAR
    Tok   : ARRAY[1..16] OF STRING;
    Codes : ARRAY[1..27] OF STRING := [
        'FF','FN','FZ','FH','FV','FO','FC','FM','FD','FQ','FS','FB','FE','FT',
        'WL','WV','WT','WS','WM','WP','WR','WH',
        'NC','NI','ND','NR','NT'
    ];
    idx, i : INT;
    flag   : STRING;
END_VAR

(* tokenise once *)
Tok := F_ZaberSplitReplyTokensEx(sInput := sInput);

(* decide flag index: if token 3 is OK/RJ → no MSG-ID *)
IF (Tok[3] = 'OK') OR (Tok[3] = 'RJ') THEN
	idx := 5;                      (* @nn 0 OK IDLE <flag> ... *)
ELSE
	idx := 6;                      (* @nn 0 01 OK IDLE <flag> ... *)
END_IF

flag := Tok[idx];

(* 1) '--' is valid and must be returned *)
IF flag = '--' THEN
	F_ZaberExtractWarnFaultFlag := '--';
	RETURN;
END_IF

(* 2) return known code if found *)
FOR i := 1 TO 27 DO
	IF flag = Codes[i] THEN
		F_ZaberExtractWarnFaultFlag := flag;
		RETURN;
	END_IF
END_FOR

(* 3) anything else → empty *)
F_ZaberExtractWarnFaultFlag := '';

END_FUNCTION

// Zaber/POUs/FB_ZaberAxisCmdConfiguration
FUNCTION_BLOCK FB_ZaberAxisCmdConfiguration EXTENDS Base.FB_BaseStatic IMPLEMENTS I_ZaberAxisConfigurationFW744, I_ZaberSerialConfiguration
VAR
	// _iFileReferenceInterface
	ZaberConfiguration					: ST_ZaberConfiguration; //NOTE ; Component and other SUPER^ REFs not defined!!!
	LocalComponentConfiguration			: Base.ST_ComponentConfiguration;
	
	ConfigStruct						: ST_ZaberInitTableFW744;
	
	LoopIndex							: DINT;
	
	ZaberCmdConfiguration				: ARRAY[GC_Zaber.INDEX_COMMAND_MIN..GC_Zaber.INDEX_COMMAND_MAX] OF Base.FB_CmdPermIntlkConfiguration;
	ipZaberCmdConfiguration				: ARRAY[GC_Zaber.INDEX_COMMAND_MIN..GC_Zaber.INDEX_COMMAND_MAX] OF I_CommandConfiguration;
	ipZaberPermIntlkConfiguration		: ARRAY[GC_Zaber.INDEX_COMMAND_MIN..GC_Zaber.INDEX_COMMAND_MAX] OF I_PermIntlkConfiguration;
	
//Hash Table
	fbHashDJB2_PouName					: Base.FB_Hash_djb2;
	iHashDJB2_PouName					: I_HashFunction := fbHashDJB2_PouName;
	
	fbHashDJB2_CmdSendString			: Base.FB_Hash_djb2;
	iHashDJB2_CmdSendString				: I_HashFunction := fbHashDJB2_CmdSendString;
	
	HashTablePouName					: Base.FB_HashTable;
	iHashTablePouName					: I_HashTableBase := HashTablePouName;
	
	HashTableCmdSendString				: Base.FB_HashTable;
	iHashTableCmdSendString				: I_HashTableBase := HashTableCmdSendString;
END_VAR

METHOD PROTECTED _BuildTables : BOOL;
FOR LoopIndex := GPL_Zaber.INDEX_COMMAND_MIN TO GPL_Zaber.INDEX_COMMAND_MAX BY 1 DO
	IF iHashTablePouName <> 0 THEN
		iHashTablePouName.Insert(IdxIn := DINT_TO_UINT(LoopIndex), NameIn := ConfigStruct.PouName[LoopIndex]);
	END_IF
	
	IF iHashTableCmdSendString <> 0 THEN
		iHashTableCmdSendString.Insert(IdxIn := DINT_TO_UINT(LoopIndex), NameIn := ConfigStruct.CmdDesc[LoopIndex]);
	END_IF
END_FOR

_BuildTables := TRUE;
END_METHOD

(* Basic component initialization logic*)
METHOD PROTECTED _Initialize : BOOL
BaseStatus.Initialized := _InitializeChildrenDependencies();

BaseStatus.Initialized	:= _InitializeReferences();

BaseStatus.Busy	:= FALSE;

IF NOT BaseStatus.Initialized THEN
	TraceWithSeverity(Message := 'Initialization Failed - look at _Initialize method', Severity := TcEventSeverity.Error);
END_IF

HashTablePouName.InjectHashFunction(iHashFunction := iHashDJB2_PouName);
HashTableCmdSendString.InjectHashFunction(iHashFunction := iHashDJB2_CmdSendString);

BaseStatus.Initialized	:= _BuildTables();

_Initialize 			:= BaseStatus.Initialized;
END_METHOD

METHOD PROTECTED _InitializeChildrenDependencies : BOOL
FOR LoopIndex := GC_Zaber.INDEX_COMMAND_MIN TO GC_Zaber.INDEX_COMMAND_MAX DO
	IF ipZaberCmdConfiguration[LoopIndex] <> 0 THEN
		ipZaberCmdConfiguration[LoopIndex].Initialize();		
	END_IF
	
	IF ipZaberPermIntlkConfiguration[LoopIndex] <> 0 THEN
		ipZaberPermIntlkConfiguration[LoopIndex].Initialize();
	END_IF
END_FOR

IF iHashDJB2_PouName <> 0 THEN
	iHashDJB2_PouName.Initialize();
END_IF

IF iHashDJB2_CmdSendString <> 0 THEN
	iHashDJB2_CmdSendString.Initialize();
END_IF

IF iHashTablePouName <> 0 THEN
	iHashTablePouName.Initialize();
END_IF

IF iHashTableCmdSendString <> 0 THEN
	iHashTableCmdSendString.Initialize();
END_IF

_InitializeChildrenDependencies := TRUE;
END_METHOD

METHOD PROTECTED _InitializeReferences : BOOL
//Order is important!
BaseConfiguration.InstancePath 	REF= SUPER^.InstancePath;

LocalComponentConfiguration.BaseConfiguration REF= SUPER^.BaseConfiguration;

ZaberConfiguration.ComponentConfiguration REF= LocalComponentConfiguration;

_InitializeReferences 			:= TRUE; // apply at end of all reference initialization
END_METHOD

//FB_Init is always available implicitly and it is used primarily for initialization.
//The return value is not evaluated. For a specific influence, you can also declare the
//methods explicitly and provide additional code there with the standard initialization
//code. You can evaluate the return value.
METHOD FB_Init: BOOL
VAR_INPUT
    bInitRetains: BOOL; // TRUE: the retain variables are initialized (reset warm / reset cold)
    bInCopyCode: BOOL;  // TRUE: the instance will be copied to the copy code afterward (online change)   
END_VAR
FOR LoopIndex := GC_Zaber.INDEX_COMMAND_MIN TO GC_Zaber.INDEX_COMMAND_MAX DO
    ipZaberCmdConfiguration[LoopIndex]       := ZaberCmdConfiguration[LoopIndex]; // implements I_CommandConfiguration
    ipZaberPermIntlkConfiguration[LoopIndex] := ZaberCmdConfiguration[LoopIndex]; // implements I_PermIntlkConfiguration
	
	ipZaberCmdConfiguration[LoopIndex].P_CommandConfiguration.CommandIndex			:= LoopIndex;
	ipZaberCmdConfiguration[LoopIndex].P_CommandConfiguration.CommandDescription	:= ConfigStruct.CmdDesc[LoopIndex];
	ipZaberCmdConfiguration[LoopIndex].P_CommandConfiguration.CommandPOUName 		:= ConfigStruct.PouName[LoopIndex];
	ipZaberCmdConfiguration[LoopIndex].P_CommandConfiguration.CommandExecutionType	:= ConfigStruct.CmdExecutionType[LoopIndex];
END_FOR
END_METHOD

//� Lookup name ? index
METHOD PUBLIC GetIndexByCmdSendString : UINT
VAR_INPUT
  NameIn : T_MaxString;
END_VAR
IF iHashTableCmdSendString <> 0 THEN
	GetIndexByCmdSendString	:= iHashTableCmdSendString.GetIndex(NameIn := NameIn);
END_IF
END_METHOD

(*� Lookup name ? index*)
METHOD GetIndexByPOUName : UINT
VAR_INPUT
	NameIn	: T_MaxString;
END_VAR
IF iHashTablePouName <> 0 THEN
	GetIndexByPOUName	:= iHashTablePouName.GetIndex(NameIn := NameIn);
END_IF
END_METHOD

PROPERTY P_CommandConfigurations : REFERENCE TO ARRAY[GC_Zaber.INDEX_COMMAND_MIN..GC_Zaber.INDEX_COMMAND_MAX] OF I_CommandConfiguration;
GET
P_CommandConfigurations REF= ipZaberCmdConfiguration;
END_GET
END_PROPERTY

PROPERTY P_PermIntlkConfigurations : REFERENCE TO ARRAY[GC_Zaber.INDEX_COMMAND_MIN..GC_Zaber.INDEX_COMMAND_MAX] OF I_PermIntlkConfiguration;
GET
P_PermIntlkConfigurations REF= ipZaberPermIntlkConfiguration;
END_GET
END_PROPERTY

PROPERTY P_ZaberConfiguration : REFERENCE TO ST_ZaberConfiguration
GET
P_ZaberConfiguration REF= ZaberConfiguration;
END_GET
END_PROPERTY

PROPERTY P_ZaberInitTableFW744 : REFERENCE TO ST_ZaberInitTableFW744
GET
P_ZaberInitTableFW744 REF= ConfigStruct;
END_GET
END_PROPERTY

END_FUNCTION_BLOCK

// Zaber/POUs/FB_ZaberSerialAxis
FUNCTION_BLOCK FB_ZaberSerialAxis EXTENDS Base.FB_Component<GC_Zaber.INDEX_COMMAND_MIN,GC_Zaber.INDEX_COMMAND_MAX> IMPLEMENTS I_ZaberSerialFW744, I_ZaberSerialConfiguration
VAR
	ZaberConfiguration				: ST_ZaberConfiguration;
	ZaberStatus						: ST_ZaberStatus;
	                            	
	PollBusyTimer					: Tc2_Standard.TON;
	WaitingForBits					: ST_WaitingForBits;
	
	_ZaberAxisConfigurationFW744	: I_ZaberAxisConfigurationFW744; // passed externally
	_ZaberSerialConfiguration		: I_ZaberSerialConfiguration;
                                	
//Serial Communication interfaces
	_iSerialTx						: Communication.I_StringCmdStatusTx;
	_iSerialRx						: Communication.I_StringCmdStatusRx;
	_iSerialConfiguration			: Communication.I_SerialConfiguration;
	_iSerialStatus					: Communication.I_SerialStatus;
	                            	
//RingBuffer	                	
	RingBufferSend					: Base.FB_RingBufferKeyString;
	iBufferSend						: Base.I_RingBufferKeyString := RingBufferSend;
                                	
	RingBufferRcv					: Base.FB_RingBufferKeyString;
	iBufferRcv						: Base.I_RingBufferKeyString := RingBufferRcv;

	RingBufferAll					: Base.FB_RingBufferKeyString;
	iBufferAll						: Base.I_RingBufferKeyString := RingBufferAll;
                                	
	ZaberCommand					: Base.ST_SystimeString;
	ZaberReceipt					: Base.ST_SystimeString;
	
	Run 		AT %I* 		: BOOL;
	ftRun					: Tc2_Standard.F_TRIG;
	
//Testing Trigs
	TrigCmd				: BOOL;
	TempPouName			: STRING;
	TempHash			: UINT;
	
//Interface test variable
	testIBufferSend		: Base.I_RingBufferKeyString;
END_VAR

METHOD comm_en_ipv4_static
VAR_INPUT
	Address : STRING := '0.0.0.0'; //The IPv4 address to use for this device must be in the range 1.0.0.0 to 223.255.255.255, or 0.0.0.0 to disable IPv4 networking
	Netmask	: STRING := '0.0.0.0'; //The IPv4 subnet mask must be in the range 255.0.0.0 to 255.255.255.254 when specified in dot-decimal notation, or in the range 8 to 31 when specified as the bit-length of the network prefix
	Gateway	: STRING := '0.0.0.0'; //The IPv4 address OF the default gateway must be in the range 1.0.0.0 TO 223.255.255.255, OR 0.0.0.0 if not using a default gateway
END_VAR
IF ZaberStatus.ComponentStatus.iLastCommand <> 0 THEN
	ZaberStatus.ComponentStatus.iLastCommand.P_CommandStatus.LastCommandMessage := Base.F_GetLastWordInString(__POUNAME());
END_IF

IF NOT _DispatchValid() THEN
	RETURN;
ELSE
	_BuildCommandStringNoArgs();
	//append additional args
	ZaberCommand.stringval := Tc2_Standard.CONCAT(STR1 := ZaberCommand.stringval, STR2 := ' ');
	ZaberCommand.stringval := Tc2_Standard.CONCAT(STR1 := ZaberCommand.stringval, STR2 := Address);
	ZaberCommand.stringval := Tc2_Standard.CONCAT(STR1 := ZaberCommand.stringval, STR2 := ' ');
	ZaberCommand.stringval := Tc2_Standard.CONCAT(STR1 := ZaberCommand.stringval, STR2 := Netmask);
	ZaberCommand.stringval := Tc2_Standard.CONCAT(STR1 := ZaberCommand.stringval, STR2 := ' ');
	ZaberCommand.stringval := Tc2_Standard.CONCAT(STR1 := ZaberCommand.stringval, STR2 := Gateway);
	
	IF iBufferSend <> 0 AND __QUERYINTERFACE(iBufferSend, testIBufferSend) THEN
		iBufferSend.AddObject(RefObject := ZaberCommand);
	END_IF	
END_IF
END_METHOD

METHOD io_cancel_schedule
IF ZaberStatus.ComponentStatus.iLastCommand <> 0 THEN
	ZaberStatus.ComponentStatus.iLastCommand.P_CommandStatus.LastCommandMessage := Base.F_GetLastWordInString(__POUNAME());
END_IF

IF NOT _DispatchValid() THEN
	RETURN;
ELSE
	_BuildCommandStringNoArgs();
	
	IF iBufferSend <> 0 AND __QUERYINTERFACE(iBufferSend, testIBufferSend) THEN
		iBufferSend.AddObject(RefObject := ZaberCommand);
	END_IF
END_IF
END_METHOD

METHOD io_set_ao
IF ZaberStatus.ComponentStatus.iLastCommand <> 0 THEN
	ZaberStatus.ComponentStatus.iLastCommand.P_CommandStatus.LastCommandMessage := Base.F_GetLastWordInString(__POUNAME());
END_IF

IF NOT _DispatchValid() THEN
	RETURN;
ELSE
	_BuildCommandStringNoArgs();
	
	IF iBufferSend <> 0 AND __QUERYINTERFACE(iBufferSend, testIBufferSend) THEN
		iBufferSend.AddObject(RefObject := ZaberCommand);
	END_IF
END_IF
END_METHOD

METHOD io_set_ao_schedule
IF ZaberStatus.ComponentStatus.iLastCommand <> 0 THEN
	ZaberStatus.ComponentStatus.iLastCommand.P_CommandStatus.LastCommandMessage := Base.F_GetLastWordInString(__POUNAME());
END_IF

IF NOT _DispatchValid() THEN
	RETURN;
ELSE
	_BuildCommandStringNoArgs();
	
	IF iBufferSend <> 0 AND __QUERYINTERFACE(iBufferSend, testIBufferSend) THEN
		iBufferSend.AddObject(RefObject := ZaberCommand);
	END_IF
END_IF
END_METHOD

METHOD io_set_do
IF ZaberStatus.ComponentStatus.iLastCommand <> 0 THEN
	ZaberStatus.ComponentStatus.iLastCommand.P_CommandStatus.LastCommandMessage := Base.F_GetLastWordInString(__POUNAME());
END_IF

IF NOT _DispatchValid() THEN
	RETURN;
ELSE
	_BuildCommandStringNoArgs();
	
	IF iBufferSend <> 0 AND __QUERYINTERFACE(iBufferSend, testIBufferSend) THEN
		iBufferSend.AddObject(RefObject := ZaberCommand);
	END_IF
END_IF
END_METHOD

METHOD io_set_do_schedule
IF ZaberStatus.ComponentStatus.iLastCommand <> 0 THEN
	ZaberStatus.ComponentStatus.iLastCommand.P_CommandStatus.LastCommandMessage := Base.F_GetLastWordInString(__POUNAME());
END_IF

IF NOT _DispatchValid() THEN
	RETURN;
ELSE
	_BuildCommandStringNoArgs();
	
	IF iBufferSend <> 0 AND __QUERYINTERFACE(iBufferSend, testIBufferSend) THEN
		iBufferSend.AddObject(RefObject := ZaberCommand);
	END_IF
END_IF
END_METHOD

METHOD lockstep_driver_disable
VAR_INPUT
	LockstepGroup	: USINT := 1; // The address of the lockstep group must be in the range 1 to lockstep.numgroups; lockstep.numgroups: the number of lockstep groupss; Valid Values: 0 to 2
END_VAR
IF ZaberStatus.ComponentStatus.iLastCommand <> 0 THEN
	ZaberStatus.ComponentStatus.iLastCommand.P_CommandStatus.LastCommandMessage := Base.F_GetLastWordInString(__POUNAME());
END_IF

IF NOT _DispatchValid() THEN
	RETURN;
ELSE
	_ClearTempString();
	ZaberCommand.stringval := Tc2_Standard.CONCAT(STR1 := ZaberConfiguration.sControllerRef, STR2 := ' ');
	ZaberCommand.stringval := Tc2_Standard.CONCAT(STR1 := ZaberCommand.stringval, STR2 := Base.F_GetFirstWordInString(sInput := SUPER^._iCommandConfiguration[ZaberStatus.ZaberMethodDispatch].P_CommandConfiguration.CommandDescription));
	ZaberCommand.stringval := Tc2_Standard.CONCAT(STR1 := ZaberCommand.stringval, STR2 := ' ');
	ZaberCommand.stringval := Tc2_Standard.CONCAT(STR1 := ZaberCommand.stringval, STR2 := USINT_TO_STRING(LockstepGroup));
	ZaberCommand.stringval := Tc2_Standard.CONCAT(STR1 := ZaberCommand.stringval, STR2 := ' ');
	ZaberCommand.stringval := Tc2_Standard.CONCAT(STR1 := ZaberCommand.stringval, STR2 := F_GetAllButFirstWord(sInput := SUPER^._iCommandConfiguration[ZaberStatus.ZaberMethodDispatch].P_CommandConfiguration.CommandDescription));
	
	IF iBufferSend <> 0 AND __QUERYINTERFACE(iBufferSend, testIBufferSend) THEN
		iBufferSend.AddObject(RefObject := ZaberCommand);
	END_IF	
END_IF
END_METHOD

METHOD lockstep_driver_enable
VAR_INPUT
	LockstepGroup	: USINT := 1; // The address of the lockstep group must be in the range 1 to lockstep.numgroups; lockstep.numgroups: the number of lockstep groupss; Valid Values: 0 to 2
END_VAR
IF ZaberStatus.ComponentStatus.iLastCommand <> 0 THEN
	ZaberStatus.ComponentStatus.iLastCommand.P_CommandStatus.LastCommandMessage := Base.F_GetLastWordInString(__POUNAME());
END_IF

